C07332=1146.015,329.799,-77.371,-176.675,8.921,148.819
C07333=1146.011,330.047,-77.404,-176.672,8.925,148.820
C07334=1146.007,330.294,-77.436,-176.670,8.928,148.820
C07335=1146.003,330.542,-77.470,-176.667,8.932,148.820
C07336=1145.999,330.789,-77.503,-176.665,8.936,148.820
C07337=1145.995,331.037,-77.536,-176.662,8.940,148.821
C07338=1145.991,331.285,-77.569,-176.659,8.943,148.821
C07339=1145.986,331.533,-77.602,-176.657,8.947,148.821
C07340=1145.982,331.780,-77.635,-176.654,8.950,148.821
C07341=1145.978,332.028,-77.669,-176.651,8.954,148.821
C07342=1145.974,332.276,-77.702,-176.649,8.958,148.822
C07343=1145.970,332.524,-77.735,-176.646,8.962,148.822
C07344=1145.966,332.771,-77.768,-176.644,8.965,148.822
C07345=1145.962,333.020,-77.802,-176.641,8.969,148.823
C07346=1145.958,333.267,-77.835,-176.639,8.973,148.823
C07347=1145.954,333.515,-77.868,-176.637,8.976,148.823
C07348=1145.950,333.763,-77.901,-176.634,8.980,148.823
C07349=1145.946,334.010,-77.935,-176.631,8.983,148.823
C07350=1145.942,334.258,-77.968,-176.628,8.987,148.824
C07351=1145.938,334.505,-78.001,-176.627,8.991,148.824
C07352=1145.934,334.753,-78.034,-176.624,8.995,148.824
C07353=1145.930,335.002,-78.068,-176.621,8.998,148.824
C07354=1145.926,335.249,-78.102,-176.618,9.002,148.825
C07355=1145.922,335.496,-78.135,-176.615,9.006,148.825
C07356=1145.918,335.744,-78.168,-176.613,9.010,148.825
C07357=1145.913,335.992,-78.202,-176.611,9.014,148.826
C07358=1145.909,336.239,-78.236,-176.608,9.017,148.826
C07359=1145.906,336.488,-78.269,-176.605,9.021,148.826
C07360=1145.902,336.735,-78.302,-176.603,9.025,148.826
C07361=1145.897,336.983,-78.336,-176.600,9.029,148.826
C07362=1145.894,337.230,-78.369,-176.598,9.032,148.827
C07363=1145.889,337.478,-78.403,-176.595,9.036,148.827
C07364=1145.885,337.727,-78.437,-176.593,9.040,148.827
C07365=1145.881,337.974,-78.471,-176.590,9.044,148.828
C07366=1145.877,338.222,-78.504,-176.588,9.047,148.828
C07367=1145.873,338.469,-78.538,-176.585,9.051,148.828
C07368=1145.869,338.716,-78.571,-176.583,9.055,148.828
C07369=1145.864,338.997,-78.609,-176.580,9.059,148.829
C07370=1145.860,339.277,-78.647,-176.577,9.064,148.829
C07371=1145.856,339.558,-78.686,-176.574,9.068,148.829
C07372=1145.851,339.839,-78.724,-176.571,9.072,148.830
C07373=1145.847,340.086,-78.757,-176.569,9.075,148.830
C07374=1145.843,340.333,-78.791,-176.566,9.080,148.830
C07375=1145.838,340.581,-78.825,-176.564,9.083,148.830
C07376=1145.835,340.829,-78.859,-176.561,9.087,148.831
C07377=1145.831,341.076,-78.893,-176.558,9.091,148.831
C07378=1145.827,341.324,-78.926,-176.556,9.095,148.831
C07379=1145.823,341.572,-78.961,-176.553,9.099,148.832
C07380=1145.819,341.820,-78.994,-176.551,9.102,148.832
C07381=1145.815,342.067,-79.028,-176.548,9.106,148.832
C07382=1145.810,342.314,-79.062,-176.546,9.110,148.832
C07383=1145.807,342.563,-79.096,-176.543,9.114,148.833
C07384=1145.802,342.810,-79.130,-176.541,9.117,148.833
C07385=1145.799,343.057,-79.164,-176.538,9.121,148.833
C07386=1145.795,343.306,-79.198,-176.536,9.126,148.834
C07387=1145.790,343.553,-79.232,-176.533,9.129,148.834
C07388=1145.787,343.800,-79.266,-176.530,9.133,148.834
C07389=1145.783,344.049,-79.300,-176.528,9.137,148.834
C07390=1145.778,344.296,-79.334,-176.525,9.141,148.835
C07391=1145.775,344.543,-79.368,-176.523,9.144,148.835
C07392=1145.771,344.791,-79.403,-176.521,9.148,148.835
C07393=1145.767,345.039,-79.436,-176.518,9.152,148.836
C07394=1145.762,345.287,-79.470,-176.515,9.156,148.836
C07395=1145.759,345.534,-79.505,-176.513,9.160,148.836
C07396=1145.754,345.782,-79.539,-176.511,9.163,148.836
C07397=1145.751,346.030,-79.573,-176.508,9.167,148.837
C07398=1145.746,346.277,-79.608,-176.506,9.171,148.837
C07399=1145.742,346.525,-79.641,-176.503,9.175,148.837
C07400=1145.738,346.773,-79.676,-176.500,9.179,148.838
C07401=1145.734,347.020,-79.710,-176.498,9.183,148.838
C07402=1145.730,347.268,-79.745,-176.495,9.187,148.838
C07403=1145.727,347.515,-79.778,-176.493,9.190,148.838
C07404=1145.722,347.763,-79.813,-176.490,9.195,148.839
C07405=1145.719,348.011,-79.847,-176.487,9.199,148.839
C07406=1145.714,348.258,-79.882,-176.485,9.202,148.839
C07407=1145.711,348.506,-79.916,-176.483,9.206,148.840
C07408=1145.706,348.753,-79.950,-176.480,9.210,148.840
C07409=1145.702,349.001,-79.985,-176.477,9.214,148.840
C07410=1145.699,349.248,-80.019,-176.475,9.217,148.841
C07411=1145.695,349.497,-80.054,-176.473,9.221,148.841
C07412=1145.691,349.744,-80.088,-176.470,9.226,148.841
C07413=1145.687,349.992,-80.123,-176.468,9.229,148.842
C07414=1145.682,350.239,-80.157,-176.465,9.233,148.842
C07415=1145.679,350.486,-80.192,-176.462,9.237,148.842
C07416=1145.675,350.734,-80.226,-176.460,9.241,148.843
C07417=1145.671,350.982,-80.261,-176.457,9.245,148.843
C07418=1145.667,351.229,-80.295,-176.455,9.248,148.843
C07419=1145.663,351.477,-80.330,-176.452,9.252,148.843
C07420=1145.658,351.725,-80.364,-176.450,9.257,148.844
C07421=1145.656,351.972,-80.399,-176.447,9.260,148.844
C07422=1145.651,352.219,-80.434,-176.445,9.264,148.845
C07423=1145.647,352.467,-80.469,-176.443,9.268,148.845
C07424=1145.643,352.714,-80.503,-176.440,9.272,148.845
C07425=1145.640,352.962,-80.538,-176.437,9.276,148.846
C07426=1145.635,353.209,-80.573,-176.435,9.279,148.846
C07427=1145.631,353.457,-80.607,-176.432,9.284,148.846
C07428=1145.627,353.704,-80.642,-176.429,9.288,148.846
C07429=1145.623,353.952,-80.677,-176.428,9.292,148.847
C07430=1145.620,354.200,-80.712,-176.425,9.296,148.847
C07431=1145.615,354.447,-80.747,-176.422,9.300,148.848
C07432=1145.612,354.695,-80.781,-176.420,9.303,148.848
C07433=1145.607,354.942,-80.816,-176.417,9.308,148.848
C07434=1145.604,355.190,-80.851,-176.415,9.311,148.848
C07435=1145.600,355.438,-80.886,-176.412,9.315,148.849
C07436=1145.596,355.685,-80.921,-176.410,9.319,148.849
C07437=1145.592,355.932,-80.955,-176.407,9.323,148.849
C07438=1145.588,356.180,-80.990,-176.405,9.327,148.850
C07439=1145.584,356.427,-81.025,-176.402,9.331,148.850
C07440=1145.580,356.675,-81.060,-176.400,9.335,148.850
C07441=1145.576,356.922,-81.095,-176.397,9.339,148.851
C07442=1145.572,357.170,-81.130,-176.394,9.343,148.851
C07443=1145.568,357.418,-81.166,-176.392,9.346,148.851
C07444=1145.564,357.665,-81.201,-176.390,9.351,148.852
C07445=1145.561,357.912,-81.235,-176.387,9.355,148.852
C07446=1145.557,358.160,-81.271,-176.385,9.359,148.853
C07447=1145.553,358.407,-81.305,-176.382,9.363,148.853
C07448=1145.549,358.655,-81.341,-176.379,9.367,148.853
C07449=1145.545,358.902,-81.376,-176.377,9.370,148.853
C07450=1145.541,359.150,-81.411,-176.375,9.375,148.854
C07451=1145.537,359.397,-81.446,-176.372,9.379,148.854
C07452=1145.533,359.645,-81.482,-176.369,9.383,148.855
C07453=1145.529,359.893,-81.517,-176.367,9.386,148.855
C07454=1145.525,360.140,-81.552,-176.364,9.391,148.855
C07455=1145.521,360.387,-81.587,-176.361,9.395,148.856
C07456=1145.517,360.635,-81.622,-176.359,9.399,148.856
C07457=1145.513,360.882,-81.657,-176.357,9.403,148.856
C07458=1145.509,361.130,-81.693,-176.354,9.407,148.857
C07459=1145.506,361.377,-81.729,-176.351,9.411,148.857
C07460=1145.502,361.625,-81.764,-176.349,9.415,148.857
C07461=1145.498,361.872,-81.799,-176.346,9.419,148.858
C07462=1145.494,362.120,-81.834,-176.343,9.423,148.858
C07463=1145.490,362.367,-81.870,-176.341,9.427,148.858
C07464=1145.487,362.615,-81.905,-176.338,9.431,148.859
C07465=1145.483,362.862,-81.941,-176.336,9.435,148.859
C07466=1145.479,363.109,-81.976,-176.333,9.439,148.859
C07467=1145.475,363.356,-82.011,-176.331,9.443,148.860
C07468=1145.471,363.604,-82.048,-176.328,9.447,148.860
C07469=1145.467,363.852,-82.082,-176.325,9.452,148.861
C07470=1145.463,364.100,-82.118,-176.322,9.456,148.861
C07471=1145.459,364.347,-82.153,-176.320,9.459,148.861
C07472=1145.455,364.594,-82.189,-176.317,9.463,148.861
C07473=1145.451,364.877,-82.230,-176.314,9.469,148.862
C07474=1145.446,365.161,-82.270,-176.311,9.473,148.862
C07475=1145.442,365.444,-82.311,-176.308,9.478,148.863
C07476=1145.437,365.728,-82.352,-176.306,9.482,148.863
C07477=1145.433,365.975,-82.388,-176.303,9.486,148.864
C07478=1145.429,366.223,-82.424,-176.300,9.491,148.864
C07479=1145.426,366.470,-82.459,-176.298,9.495,148.864
C07480=1145.422,366.717,-82.495,-176.295,9.499,148.865
C07481=1145.419,366.965,-82.531,-176.292,9.503,148.865
C07482=1145.414,367.213,-82.567,-176.290,9.508,148.865
C07483=1145.410,367.459,-82.602,-176.287,9.512,148.866
C07484=1145.406,367.707,-82.638,-176.284,9.516,148.866
C07485=1145.402,367.955,-82.674,-176.282,9.519,148.866
C07486=1145.399,368.202,-82.710,-176.279,9.524,148.867
C07487=1145.395,368.449,-82.746,-176.277,9.528,148.867
C07488=1145.390,368.697,-82.782,-176.274,9.532,148.868
C07489=1145.387,368.944,-82.817,-176.271,9.537,148.868
C07490=1145.383,369.191,-82.854,-176.269,9.541,148.869
C07491=1145.379,369.439,-82.890,-176.266,9.545,148.869
C07492=1145.375,369.687,-82.925,-176.264,9.550,148.869
C07493=1145.372,369.934,-82.961,-176.261,9.554,148.870
C07494=1145.368,370.181,-82.998,-176.259,9.557,148.870
C07495=1145.363,370.428,-83.033,-176.256,9.562,148.870
C07496=1145.360,370.675,-83.069,-176.254,9.566,148.871
C07497=1145.356,370.923,-83.105,-176.251,9.570,148.871
C07498=1145.352,371.170,-83.141,-176.248,9.575,148.872
C07499=1145.348,371.417,-83.178,-176.246,9.579,148.872
C07500=1145.344,371.665,-83.213,-176.243,9.583,148.873
C07501=1145.341,371.912,-83.250,-176.241,9.587,148.873
C07502=1145.336,372.160,-83.286,-176.238,9.591,148.873
C07503=1145.333,372.407,-83.322,-176.236,9.595,148.874
C07504=1145.329,372.654,-83.358,-176.233,9.600,148.874
C07505=1145.325,372.901,-83.394,-176.231,9.604,148.875
C07506=1145.321,373.149,-83.431,-176.228,9.608,148.875
C07507=1145.318,373.396,-83.467,-176.227,9.612,148.876
C07508=1145.313,373.644,-83.503,-176.224,9.616,148.876
C07509=1145.310,373.891,-83.539,-176.222,9.621,148.876
C07510=1145.305,374.138,-83.575,-176.219,9.625,148.877
C07511=1145.303,374.386,-83.612,-176.217,9.629,148.877
C07512=1145.298,374.634,-83.648,-176.215,9.633,148.878
C07513=1145.295,374.881,-83.684,-176.212,9.638,148.878
C07514=1145.291,375.128,-83.721,-176.210,9.641,148.879
C07515=1145.287,375.375,-83.757,-176.208,9.646,148.879
C07516=1145.283,375.623,-83.794,-176.205,9.650,148.880
C07517=1145.279,375.870,-83.831,-176.204,9.654,148.880
C07518=1145.275,376.117,-83.866,-176.201,9.658,148.881
C07519=1145.271,376.364,-83.903,-176.199,9.662,148.881
C07520=1145.268,376.611,-83.939,-176.197,9.666,148.882
C07521=1145.264,376.859,-83.976,-176.195,9.670,148.882
C07522=1145.259,377.106,-84.012,-176.193,9.674,148.883
C07523=1145.256,377.353,-84.048,-176.191,9.678,148.883
C07524=1145.253,377.601,-84.086,-176.189,9.683,148.884
C07525=1145.248,377.848,-84.123,-176.187,9.686,148.884
C07526=1145.245,378.095,-84.159,-176.185,9.691,148.885
C07527=1145.241,378.343,-84.195,-176.183,9.695,148.886
C07528=1145.237,378.590,-84.232,-176.181,9.698,148.886
C07529=1145.233,378.837,-84.268,-176.180,9.702,148.887
C07530=1145.229,379.084,-84.305,-176.178,9.707,148.887
C07531=1145.225,379.331,-84.342,-176.176,9.711,148.888
C07532=1145.222,379.579,-84.378,-176.174,9.714,148.888
C07533=1145.218,379.826,-84.415,-176.173,9.718,148.889
C07534=1145.214,380.074,-84.451,-176.171,9.722,148.889
C07535=1145.210,380.321,-84.488,-176.170,9.726,148.890
C07536=1145.206,380.568,-84.525,-176.168,9.730,148.891
C07537=1145.202,380.815,-84.561,-176.167,9.734,148.891
C07538=1145.199,381.063,-84.599,-176.165,9.738,148.892
C07539=1145.195,381.310,-84.635,-176.164,9.742,148.893
C07540=1145.191,381.557,-84.672,-176.162,9.746,148.893
C07541=1145.187,381.804,-84.709,-176.162,9.749,148.894
C07542=1145.183,382.052,-84.745,-176.160,9.752,148.894
C07543=1145.179,382.299,-84.782,-176.159,9.757,148.895
C07544=1145.176,382.546,-84.819,-176.158,9.760,148.896
C07545=1145.172,382.794,-84.856,-176.157,9.764,148.896
C07546=1145.168,383.041,-84.893,-176.156,9.767,148.897
C07547=1145.164,383.288,-84.930,-176.155,9.770,148.898
C07548=1145.160,383.535,-84.966,-176.154,9.774,148.898
C07549=1145.157,383.783,-85.003,-176.153,9.777,148.899
C07550=1145.153,384.029,-85.041,-176.153,9.781,148.900
C07551=1145.149,384.277,-85.077,-176.152,9.784,148.900
C07552=1145.145,384.524,-85.114,-176.152,9.787,148.901
C07553=1145.142,384.772,-85.152,-176.151,9.791,148.902
C07554=1145.138,385.019,-85.188,-176.150,9.794,148.903
C07555=1145.134,385.266,-85.225,-176.150,9.797,148.903
C07556=1145.130,385.513,-85.261,-176.149,9.801,148.904
C07557=1145.126,385.760,-85.298,-176.149,9.804,148.905
C07558=1145.123,386.008,-85.336,-176.149,9.807,148.906
C07559=1145.119,386.255,-85.373,-176.148,9.810,148.906
C07560=1145.115,386.502,-85.410,-176.149,9.813,148.907
C07561=1145.111,386.749,-85.446,-176.148,9.816,148.908
C07562=1145.108,386.996,-85.483,-176.149,9.819,148.909
C07563=1145.104,387.244,-85.520,-176.149,9.821,148.909
C07564=1145.100,387.491,-85.557,-176.149,9.825,148.910
C07565=1145.096,387.737,-85.595,-176.149,9.828,148.911
C07566=1145.092,387.985,-85.632,-176.149,9.830,148.912
C07567=1145.088,388.233,-85.669,-176.149,9.833,148.913
C07568=1145.084,388.480,-85.706,-176.149,9.836,148.913
C07569=1145.081,388.727,-85.742,-176.150,9.838,148.914
C07570=1145.078,388.974,-85.780,-176.150,9.841,148.915
C07571=1145.073,389.221,-85.817,-176.151,9.844,148.916
C07572=1145.069,389.468,-85.854,-176.151,9.846,148.916
C07573=1145.066,389.716,-85.891,-176.151,9.849,148.917
C07574=1145.062,389.963,-85.928,-176.152,9.852,148.918
C07575=1145.058,390.210,-85.965,-176.152,9.855,148.919
C07576=1145.054,390.457,-86.002,-176.152,9.858,148.920
C07577=1145.050,390.745,-86.045,-176.153,9.860,148.921
C07578=1145.046,391.031,-86.088,-176.154,9.863,148.922
C07579=1145.041,391.318,-86.131,-176.155,9.866,148.923
C07580=1145.037,391.605,-86.174,-176.155,9.869,148.924
C07581=1145.033,391.852,-86.211,-176.156,9.872,148.924
C07582=1145.029,392.099,-86.248,-176.157,9.874,148.925
C07583=1145.026,392.347,-86.285,-176.157,9.876,148.926
C07584=1145.022,392.594,-86.322,-176.159,9.879,148.927
C07585=1145.018,392.841,-86.360,-176.160,9.881,148.928
C07586=1145.014,393.088,-86.397,-176.160,9.883,148.929
C07587=1145.010,393.336,-86.434,-176.161,9.885,148.929
C07588=1145.006,393.583,-86.471,-176.162,9.887,148.930
C07589=1145.002,393.830,-86.508,-176.162,9.890,148.931
C07590=1145.000,394.077,-86.545,-176.164,9.892,148.932
C07591=1144.995,394.324,-86.582,-176.165,9.894,148.933
C07592=1144.991,394.571,-86.619,-176.166,9.896,148.934
C07593=1144.988,394.818,-86.656,-176.166,9.899,148.934
C07594=1144.984,395.066,-86.693,-176.167,9.901,148.935
C07595=1144.980,395.313,-86.730,-176.168,9.903,148.936
C07596=1144.976,395.560,-86.767,-176.170,9.905,148.937
C07597=1144.972,395.807,-86.805,-176.171,9.907,148.938
C07598=1144.969,396.055,-86.842,-176.172,9.910,148.939
C07599=1144.965,396.302,-86.879,-176.173,9.912,148.939
C07600=1144.960,396.549,-86.916,-176.174,9.914,148.940
C07601=1144.957,396.796,-86.954,-176.175,9.916,148.941
C07602=1144.953,397.044,-86.990,-176.176,9.918,148.942
C07603=1144.949,397.291,-87.027,-176.177,9.920,148.943
C07604=1144.945,397.538,-87.064,-176.178,9.922,148.944
C07605=1144.943,397.785,-87.101,-176.179,9.924,148.944
C07606=1144.938,398.032,-87.138,-176.181,9.926,148.945
C07607=1144.934,398.279,-87.175,-176.182,9.928,148.946
C07608=1144.931,398.527,-87.212,-176.183,9.930,148.947
C07609=1144.927,398.774,-87.250,-176.184,9.932,148.948
C07610=1144.923,399.021,-87.287,-176.185,9.934,148.949
C07611=1144.919,399.268,-87.324,-176.186,9.936,148.950
C07612=1144.916,399.515,-87.362,-176.187,9.938,148.950
C07613=1144.912,399.763,-87.398,-176.188,9.940,148.951
C07614=1144.907,400.010,-87.435,-176.190,9.942,148.952
C07615=1144.903,400.257,-87.472,-176.191,9.944,148.953
C07616=1144.900,400.504,-87.510,-176.192,9.946,148.954
C07617=1144.896,400.751,-87.547,-176.193,9.948,148.954
C07618=1144.892,400.999,-87.584,-176.194,9.950,148.955
C07619=1144.889,401.247,-87.621,-176.195,9.952,148.956
C07620=1144.885,401.493,-87.658,-176.196,9.954,148.957
C07621=1144.881,401.740,-87.695,-176.198,9.956,148.958
C07622=1144.877,401.987,-87.732,-176.199,9.957,148.959
C07623=1144.874,402.235,-87.769,-176.200,9.959,148.959
C07624=1144.870,402.482,-87.807,-176.201,9.961,148.960
C07625=1144.866,402.729,-87.843,-176.203,9.964,148.961
C07626=1144.862,402.976,-87.880,-176.203,9.965,148.962
C07627=1144.858,403.224,-87.918,-176.204,9.967,148.963
C07628=1144.855,403.471,-87.955,-176.206,9.969,148.963
C07629=1144.850,403.718,-87.992,-176.207,9.971,148.964
C07630=1144.847,403.966,-88.029,-176.208,9.973,148.965
C07631=1144.843,404.213,-88.066,-176.209,9.975,148.966
C07632=1144.839,404.459,-88.104,-176.210,9.977,148.967
C07633=1144.835,404.707,-88.140,-176.211,9.979,148.967
C07634=1144.831,404.954,-88.178,-176.213,9.981,148.968
C07635=1144.828,405.201,-88.215,-176.213,9.983,148.969
C07636=1144.824,405.448,-88.252,-176.215,9.984,148.970
C07637=1144.821,405.696,-88.289,-176.216,9.986,148.971
C07638=1144.817,405.943,-88.326,-176.217,9.988,148.971
C07639=1144.813,406.190,-88.363,-176.218,9.990,148.972
C07640=1144.809,406.437,-88.400,-176.219,9.992,148.973
C07641=1144.805,406.685,-88.437,-176.220,9.994,148.974
C07642=1144.801,406.932,-88.474,-176.221,9.996,148.975
C07643=1144.797,407.178,-88.512,-176.222,9.998,148.975
C07644=1144.793,407.426,-88.549,-176.223,10.000,148.976
C07645=1144.790,407.673,-88.586,-176.224,10.002,148.977
C07646=1144.786,407.921,-88.623,-176.226,10.003,148.978
C07647=1144.782,408.167,-88.660,-176.227,10.005,148.978
C07648=1144.779,408.415,-88.697,-176.228,10.007,148.979
C07649=1144.775,408.662,-88.734,-176.228,10.009,148.980
C07650=1144.771,408.909,-88.771,-176.229,10.011,148.981
C07651=1144.767,409.156,-88.808,-176.231,10.013,148.982
C07652=1144.764,409.404,-88.845,-176.231,10.015,148.982
C07653=1144.760,409.651,-88.882,-176.232,10.017,148.983
C07654=1144.756,409.897,-88.920,-176.233,10.019,148.984
C07655=1144.752,410.145,-88.957,-176.234,10.021,148.985
C07656=1144.748,410.392,-88.994,-176.235,10.023,148.985
C07657=1144.744,410.640,-89.031,-176.236,10.025,148.986
C07658=1144.740,410.886,-89.068,-176.237,10.027,148.987
C07659=1144.737,411.134,-89.106,-176.238,10.029,148.988
C07660=1144.733,411.381,-89.142,-176.238,10.031,148.988
C07661=1144.729,411.629,-89.179,-176.239,10.033,148.989
C07662=1144.725,411.875,-89.217,-176.240,10.035,148.990
C07663=1144.721,412.123,-89.254,-176.241,10.037,148.991
C07664=1144.717,412.370,-89.291,-176.242,10.039,148.991
C07665=1144.713,412.617,-89.328,-176.243,10.041,148.992
C07666=1144.710,412.865,-89.366,-176.244,10.043,148.993
C07667=1144.707,413.112,-89.402,-176.244,10.045,148.994
C07668=1144.703,413.359,-89.439,-176.245,10.047,148.994
C07669=1144.699,413.605,-89.476,-176.246,10.049,148.995
C07670=1144.695,413.853,-89.514,-176.247,10.052,148.996
C07671=1144.691,414.100,-89.550,-176.247,10.053,148.997
C07672=1144.687,414.348,-89.587,-176.248,10.055,148.997
C07673=1144.684,414.595,-89.625,-176.249,10.057,148.998
C07674=1144.680,414.842,-89.662,-176.250,10.059,148.999
C07675=1144.677,415.089,-89.699,-176.250,10.062,149.000
C07676=1144.676,415.337,-89.736,-176.251,10.064,149.000
C07677=1144.675,415.580,-89.772,-176.252,10.066,149.001
C07678=1144.675,415.824,-89.809,-176.253,10.067,149.002
C07679=1144.675,416.068,-89.845,-176.253,10.069,149.002
C07680=1144.676,416.312,-89.881,-176.253,10.072,149.003
C07681=1144.677,416.555,-89.916,-176.254,10.073,149.004
C07682=1144.679,416.799,-89.953,-176.255,10.075,149.004
C07683=1144.682,417.042,-89.989,-176.256,10.077,149.005
C07684=1144.686,417.285,-90.024,-176.256,10.079,149.006
C07685=1144.266,417.287,-90.074,-176.258,10.090,149.009
C07686=1144.263,417.042,-90.038,-176.257,10.088,149.008
C07687=1144.259,416.797,-90.002,-176.257,10.086,149.008
C07688=1144.256,416.552,-89.966,-176.257,10.084,149.007
C07689=1144.255,416.307,-89.929,-176.256,10.082,149.006
C07690=1144.254,416.062,-89.893,-176.255,10.081,149.006
C07691=1144.254,415.816,-89.857,-176.254,10.079,149.005
C07692=1144.254,415.571,-89.821,-176.253,10.077,149.004
C07693=1144.255,415.325,-89.784,-176.253,10.074,149.004
C07694=1144.258,415.078,-89.747,-176.252,10.072,149.003
C07695=1144.260,414.831,-89.710,-176.252,10.070,149.002
C07696=1144.263,414.583,-89.673,-176.251,10.068,149.001
C07697=1144.267,414.336,-89.636,-176.250,10.067,149.001
C07698=1144.270,414.089,-89.598,-176.249,10.064,149.000
C07699=1144.274,413.842,-89.561,-176.249,10.062,148.999
C07700=1144.278,413.594,-89.525,-176.248,10.060,148.998
C07701=1144.282,413.347,-89.487,-176.247,10.058,148.998
C07702=1144.286,413.100,-89.450,-176.246,10.056,148.997
C07703=1144.290,412.853,-89.413,-176.245,10.054,148.996
C07704=1144.294,412.606,-89.375,-176.245,10.051,148.995
C07705=1144.297,412.358,-89.338,-176.244,10.050,148.995
C07706=1144.301,412.111,-89.301,-176.243,10.048,148.994
C07707=1144.305,411.864,-89.264,-176.242,10.046,148.993
C07708=1144.308,411.617,-89.226,-176.241,10.044,148.992
C07709=1144.313,411.369,-89.190,-176.240,10.042,148.992
C07710=1144.317,411.122,-89.153,-176.240,10.040,148.991
C07711=1144.320,410.876,-89.115,-176.238,10.038,148.990
C07712=1144.323,410.628,-89.079,-176.237,10.036,148.989
C07713=1144.327,410.381,-89.042,-176.237,10.034,148.989
C07714=1144.331,410.134,-89.005,-176.236,10.032,148.988
C07715=1144.335,409.886,-88.967,-176.235,10.030,148.987
C07716=1144.339,409.639,-88.930,-176.234,10.028,148.986
C07717=1144.343,409.392,-88.893,-176.233,10.026,148.986
C07718=1144.347,409.145,-88.856,-176.232,10.024,148.985
C07719=1144.350,408.898,-88.818,-176.231,10.022,148.984
C07720=1144.354,408.650,-88.782,-176.230,10.020,148.983
C07721=1144.358,408.403,-88.745,-176.229,10.018,148.982
C07722=1144.361,408.156,-88.707,-176.228,10.016,148.982
C07723=1144.366,407.909,-88.670,-176.227,10.014,148.981
C07724=1144.370,407.662,-88.633,-176.226,10.012,148.980
C07725=1144.374,407.414,-88.596,-176.225,10.010,148.979
C07726=1144.377,407.167,-88.558,-176.224,10.008,148.978
C07727=1144.381,406.920,-88.521,-176.223,10.006,148.978
C07728=1144.385,406.673,-88.485,-176.222,10.004,148.977
C07729=1144.389,406.426,-88.447,-176.221,10.002,148.976
C07730=1144.392,406.179,-88.410,-176.220,10.000,148.975
C07731=1144.396,405.931,-88.373,-176.218,9.999,148.975
C07732=1144.400,405.684,-88.337,-176.217,9.997,148.974
C07733=1144.403,405.437,-88.299,-176.216,9.995,148.973
C07734=1144.407,405.190,-88.262,-176.215,9.993,148.972
C07735=1144.411,404.942,-88.225,-176.214,9.991,148.971
C07736=1144.415,404.695,-88.188,-176.213,9.989,148.971
C07737=1144.418,404.448,-88.150,-176.212,9.987,148.970
C07738=1144.423,404.201,-88.113,-176.211,9.985,148.969
C07739=1144.427,403.954,-88.076,-176.209,9.984,148.968
C07740=1144.430,403.706,-88.038,-176.208,9.982,148.967
C07741=1144.434,403.459,-88.002,-176.207,9.979,148.966
C07742=1144.438,403.212,-87.965,-176.206,9.977,148.966
C07743=1144.442,402.965,-87.928,-176.205,9.976,148.965
C07744=1144.445,402.718,-87.890,-176.204,9.974,148.964
C07745=1144.449,402.470,-87.853,-176.203,9.972,148.963
C07746=1144.453,402.223,-87.817,-176.202,9.970,148.963
C07747=1144.456,401.976,-87.780,-176.200,9.968,148.962
C07748=1144.460,401.729,-87.742,-176.199,9.966,148.961
C07749=1144.464,401.482,-87.705,-176.198,9.964,148.960
C07750=1144.468,401.235,-87.668,-176.197,9.962,148.959
C07751=1144.471,400.987,-87.630,-176.196,9.960,148.958
C07752=1144.476,400.740,-87.594,-176.194,9.959,148.958
C07753=1144.480,400.493,-87.557,-176.193,9.957,148.957
C07754=1144.483,400.245,-87.519,-176.192,9.955,148.956
C07755=1144.487,399.999,-87.482,-176.191,9.953,148.955
C07756=1144.491,399.751,-87.445,-176.190,9.950,148.954
C07757=1144.495,399.504,-87.408,-176.189,9.948,148.953
C07758=1144.499,399.256,-87.371,-176.188,9.946,148.953
C07759=1144.502,399.010,-87.333,-176.187,9.944,148.952
C07760=1144.506,398.762,-87.297,-176.186,9.942,148.951
C07761=1144.510,398.515,-87.259,-176.184,9.941,148.950
C07762=1144.514,398.268,-87.222,-176.183,9.939,148.949
C07763=1144.518,398.021,-87.185,-176.182,9.937,148.948
C07764=1144.521,397.774,-87.149,-176.181,9.935,148.948
C07765=1144.525,397.526,-87.111,-176.180,9.933,148.947
C07766=1144.528,397.279,-87.074,-176.178,9.931,148.946
C07767=1144.533,397.032,-87.037,-176.177,9.929,148.945
C07768=1144.537,396.785,-87.000,-176.176,9.927,148.944
C07769=1144.540,396.537,-86.963,-176.175,9.924,148.943
C07770=1144.544,396.291,-86.925,-176.174,9.922,148.943
C07771=1144.548,396.043,-86.888,-176.173,9.920,148.942
C07772=1144.552,395.796,-86.851,-176.172,9.918,148.941
C07773=1144.555,395.549,-86.814,-176.171,9.916,148.940
C07774=1144.559,395.302,-86.777,-176.170,9.913,148.939
C07775=1144.563,395.055,-86.740,-176.169,9.911,148.938
C07776=1144.567,394.807,-86.703,-176.168,9.909,148.938
C07777=1144.571,394.560,-86.665,-176.167,9.907,148.937
C07778=1144.575,394.313,-86.628,-176.166,9.905,148.936
C07779=1144.578,394.065,-86.591,-176.165,9.903,148.935
C07780=1144.582,393.818,-86.554,-176.164,9.900,148.934
C07781=1144.586,393.572,-86.517,-176.163,9.898,148.933
C07782=1144.590,393.324,-86.480,-176.162,9.896,148.933
C07783=1144.593,393.077,-86.443,-176.162,9.893,148.932
C07784=1144.597,392.830,-86.406,-176.160,9.891,148.931
C07785=1144.601,392.583,-86.369,-176.159,9.889,148.930
C07786=1144.604,392.335,-86.331,-176.159,9.887,148.929
C07787=1144.609,392.088,-86.295,-176.158,9.884,148.928
C07788=1144.612,391.841,-86.257,-176.158,9.882,148.928
C07789=1144.616,391.594,-86.220,-176.157,9.880,148.927
C07790=1144.620,391.306,-86.177,-176.156,9.877,148.926
C07791=1144.625,391.020,-86.134,-176.155,9.873,148.925
C07792=1144.629,390.733,-86.091,-176.155,9.871,148.924
C07793=1144.634,390.445,-86.048,-176.154,9.868,148.923
C07794=1144.637,390.199,-86.011,-176.153,9.866,148.922
C07795=1144.641,389.951,-85.974,-176.153,9.863,148.921
C07796=1144.645,389.704,-85.937,-176.152,9.860,148.921
C07797=1144.649,389.457,-85.900,-176.152,9.857,148.920
C07798=1144.653,389.210,-85.863,-176.152,9.855,148.919
C07799=1144.656,388.962,-85.825,-176.151,9.852,148.918
C07800=1144.660,388.715,-85.789,-176.151,9.849,148.917
C07801=1144.664,388.468,-85.752,-176.151,9.846,148.916
C07802=1144.668,388.221,-85.715,-176.151,9.844,148.916
C07803=1144.672,387.974,-85.677,-176.150,9.841,148.915
C07804=1144.675,387.727,-85.641,-176.150,9.838,148.914
C07805=1144.679,387.480,-85.604,-176.150,9.836,148.913
C07806=1144.683,387.232,-85.567,-176.150,9.832,148.913
C07807=1144.687,386.984,-85.530,-176.150,9.830,148.912
C07808=1144.690,386.738,-85.492,-176.150,9.827,148.911
C07809=1144.694,386.491,-85.455,-176.150,9.824,148.910
C07810=1144.699,386.243,-85.418,-176.150,9.821,148.910
C07811=1144.701,385.996,-85.382,-176.151,9.818,148.909
C07812=1144.705,385.749,-85.345,-176.151,9.814,148.908
C07813=1144.709,385.502,-85.308,-176.151,9.812,148.907
C07814=1144.714,385.254,-85.271,-176.151,9.808,148.907
C07815=1144.717,385.007,-85.233,-176.152,9.805,148.906
C07816=1144.721,384.760,-85.196,-176.152,9.802,148.905
C07817=1144.725,384.513,-85.160,-176.153,9.798,148.904
C07818=1144.728,384.266,-85.123,-176.153,9.795,148.904
C07819=1144.732,384.018,-85.086,-176.154,9.792,148.903
C07820=1144.736,383.771,-85.049,-176.155,9.789,148.902
C07821=1144.740,383.524,-85.012,-176.155,9.785,148.902
C07822=1144.744,383.276,-84.975,-176.157,9.781,148.901
C07823=1144.748,383.029,-84.939,-176.157,9.778,148.900
C07824=1144.751,382.782,-84.902,-176.158,9.775,148.900
C07825=1144.755,382.535,-84.864,-176.160,9.771,148.899
C07826=1144.759,382.288,-84.828,-176.160,9.768,148.898
C07827=1144.763,382.041,-84.791,-176.162,9.764,148.898
C07828=1144.766,381.793,-84.754,-176.163,9.760,148.897
C07829=1144.770,381.546,-84.717,-176.164,9.757,148.897
C07830=1144.774,381.299,-84.680,-176.166,9.753,148.896
C07831=1144.778,381.051,-84.643,-176.167,9.749,148.895
C07832=1144.782,380.804,-84.607,-176.168,9.745,148.894
C07833=1144.785,380.557,-84.570,-176.170,9.741,148.894
C07834=1144.789,380.309,-84.534,-176.172,9.737,148.893
C07835=1144.793,380.062,-84.497,-176.173,9.733,148.893
C07836=1144.797,379.815,-84.461,-176.175,9.730,148.892
C07837=1144.801,379.568,-84.424,-176.176,9.726,148.892
C07838=1144.805,379.320,-84.387,-176.178,9.722,148.891
C07839=1144.809,379.073,-84.350,-176.180,9.718,148.891
C07840=1144.812,378.826,-84.314,-176.182,9.714,148.890
C07841=1144.816,378.578,-84.277,-176.183,9.710,148.889
C07842=1144.820,378.331,-84.240,-176.185,9.706,148.889
C07843=1144.824,378.084,-84.204,-176.187,9.701,148.888
C07844=1144.828,377.837,-84.167,-176.189,9.698,148.888
C07845=1144.832,377.589,-84.131,-176.191,9.694,148.887
C07846=1144.835,377.343,-84.094,-176.193,9.690,148.887
C07847=1144.839,377.095,-84.057,-176.194,9.686,148.886
C07848=1144.844,376.848,-84.021,-176.197,9.681,148.886
C07849=1144.846,376.600,-83.985,-176.199,9.678,148.885
C07850=1144.850,376.353,-83.948,-176.201,9.673,148.885
C07851=1144.855,376.106,-83.911,-176.203,9.669,148.884
C07852=1144.858,375.858,-83.875,-176.205,9.665,148.884
C07853=1144.862,375.611,-83.839,-176.208,9.661,148.883
C07854=1144.866,375.364,-83.802,-176.210,9.657,148.883
C07855=1144.870,375.116,-83.766,-176.212,9.652,148.882
C07856=1144.873,374.869,-83.730,-176.214,9.648,148.882
C07857=1144.878,374.622,-83.693,-176.216,9.644,148.881
C07858=1144.881,374.375,-83.657,-176.219,9.640,148.881
C07859=1144.885,374.127,-83.621,-176.221,9.636,148.880
C07860=1144.889,373.880,-83.584,-176.223,9.632,148.880
C07861=1144.893,373.633,-83.548,-176.226,9.628,148.879
C07862=1144.897,373.386,-83.511,-176.228,9.623,148.879
C07863=1144.901,373.138,-83.476,-176.231,9.619,148.878
C07864=1144.905,372.891,-83.439,-176.233,9.615,148.878
C07865=1144.909,372.643,-83.403,-176.236,9.611,148.878
C07866=1144.912,372.396,-83.367,-176.238,9.607,148.877
C07867=1144.916,372.149,-83.331,-176.241,9.602,148.877
C07868=1144.920,371.902,-83.295,-176.243,9.598,148.876
C07869=1144.924,371.654,-83.259,-176.246,9.594,148.876
C07870=1144.927,371.407,-83.222,-176.249,9.590,148.876
C07871=1144.932,371.159,-83.186,-176.250,9.586,148.875
C07872=1144.935,370.912,-83.150,-176.253,9.582,148.875
C07873=1144.940,370.665,-83.114,-176.255,9.577,148.874
C07874=1144.943,370.417,-83.078,-176.258,9.573,148.874
C07875=1144.947,370.170,-83.042,-176.261,9.569,148.874
C07876=1144.951,369.922,-83.006,-176.263,9.564,148.873
C07877=1144.955,369.675,-82.970,-176.266,9.560,148.873
C07878=1144.958,369.428,-82.934,-176.269,9.556,148.872
C07879=1144.962,369.180,-82.898,-176.271,9.552,148.872
C07880=1144.966,368.933,-82.862,-176.274,9.548,148.872
C07881=1144.969,368.686,-82.826,-176.276,9.544,148.871
C07882=1144.974,368.438,-82.790,-176.279,9.539,148.871
C07883=1144.977,368.190,-82.754,-176.282,9.535,148.870
C07884=1144.981,367.943,-82.719,-176.284,9.531,148.870
C07885=1144.986,367.695,-82.683,-176.287,9.527,148.870
C07886=1144.990,367.449,-82.647,-176.289,9.523,148.869
C07887=1144.993,367.202,-82.611,-176.292,9.518,148.869
C07888=1144.998,366.954,-82.575,-176.295,9.514,148.869
C07889=1145.001,366.706,-82.539,-176.297,9.510,148.868
C07890=1145.005,366.459,-82.504,-176.300,9.506,148.868
C07891=1145.009,366.211,-82.468,-176.302,9.502,148.867
C07892=1145.013,365.963,-82.432,-176.305,9.498,148.867
C07893=1145.017,365.717,-82.396,-176.308,9.494,148.867
C07894=1145.021,365.433,-82.355,-176.311,9.489,148.866
C07895=1145.025,365.149,-82.315,-176.314,9.484,148.866
C07896=1145.030,364.866,-82.274,-176.317,9.479,148.866
C07897=1145.034,364.582,-82.234,-176.320,9.475,148.865
C07898=1145.038,364.335,-82.198,-176.322,9.471,148.865
C07899=1145.042,364.088,-82.163,-176.325,9.467,148.864
C07900=1145.046,363.841,-82.127,-176.328,9.462,148.864
C07901=1145.050,363.593,-82.091,-176.331,9.458,148.864
C07902=1145.054,363.345,-82.056,-176.333,9.454,148.863
C07903=1145.058,363.098,-82.020,-176.335,9.450,148.863
C07904=1145.061,362.850,-81.985,-176.338,9.446,148.862
C07905=1145.066,362.603,-81.949,-176.341,9.442,148.862
C07906=1145.069,362.356,-81.914,-176.343,9.438,148.862
C07907=1145.073,362.108,-81.878,-176.346,9.433,148.861
C07908=1145.077,361.860,-81.843,-176.348,9.430,148.861
C07909=1145.081,361.614,-81.808,-176.351,9.426,148.861
C07910=1145.085,361.366,-81.773,-176.354,9.422,148.861
C07911=1145.088,361.119,-81.737,-176.356,9.417,148.860
C07912=1145.092,360.871,-81.702,-176.359,9.414,148.860
C07913=1145.097,360.624,-81.667,-176.361,9.410,148.859
C07914=1145.100,360.376,-81.632,-176.364,9.406,148.859
C07915=1145.104,360.129,-81.596,-176.367,9.401,148.859
C07916=1145.108,359.881,-81.560,-176.369,9.398,148.858
C07917=1145.112,359.634,-81.526,-176.372,9.394,148.858
C07918=1145.116,359.386,-81.490,-176.374,9.389,148.858
C07919=1145.120,359.139,-81.455,-176.377,9.385,148.857
C07920=1145.124,358.891,-81.420,-176.379,9.382,148.857
C07921=1145.128,358.644,-81.385,-176.382,9.377,148.857
C07922=1145.131,358.396,-81.349,-176.385,9.373,148.856
C07923=1145.135,358.148,-81.315,-176.387,9.370,148.856
C07924=1145.140,357.901,-81.279,-176.390,9.366,148.856
C07925=1145.144,357.653,-81.245,-176.392,9.361,148.855
C07926=1145.147,357.406,-81.209,-176.394,9.358,148.855
C07927=1145.152,357.159,-81.174,-176.397,9.354,148.855
C07928=1145.155,356.911,-81.140,-176.400,9.350,148.854
C07929=1145.159,356.664,-81.104,-176.402,9.346,148.854
C07930=1145.163,356.416,-81.070,-176.405,9.342,148.854
C07931=1145.167,356.169,-81.034,-176.407,9.338,148.853
C07932=1145.171,355.921,-81.000,-176.409,9.334,148.853
C07933=1145.175,355.674,-80.964,-176.412,9.330,148.853
C07934=1145.179,355.426,-80.929,-176.415,9.326,148.852
C07935=1145.183,355.179,-80.895,-176.417,9.322,148.852
C07936=1145.186,354.931,-80.860,-176.420,9.318,148.852
C07937=1145.191,354.684,-80.825,-176.422,9.314,148.851
C07938=1145.195,354.436,-80.790,-176.424,9.310,148.851
C07939=1145.199,354.188,-80.755,-176.427,9.306,148.850
C07940=1145.202,353.941,-80.721,-176.430,9.302,148.850
C07941=1145.206,353.693,-80.685,-176.432,9.298,148.850
C07942=1145.211,353.446,-80.651,-176.435,9.294,148.850
C07943=1145.215,353.198,-80.616,-176.438,9.290,148.849
C07944=1145.218,352.951,-80.582,-176.440,9.287,148.849
C07945=1145.222,352.703,-80.547,-176.442,9.283,148.849
C07946=1145.226,352.455,-80.512,-176.444,9.279,148.848
C07947=1145.231,352.208,-80.477,-176.447,9.275,148.848
C07948=1145.234,351.961,-80.442,-176.450,9.271,148.847
C07949=1145.238,351.713,-80.408,-176.452,9.267,148.847
C07950=1145.242,351.465,-80.373,-176.455,9.263,148.847
C07951=1145.246,351.218,-80.339,-176.458,9.259,148.847
C07952=1145.250,350.970,-80.304,-176.460,9.256,148.846
C07953=1145.254,350.723,-80.269,-176.462,9.251,148.846
C07954=1145.257,350.475,-80.235,-176.465,9.248,148.846
C07955=1145.262,350.228,-80.201,-176.467,9.243,148.845
C07956=1145.266,349.980,-80.166,-176.470,9.239,148.845
C07957=1145.270,349.733,-80.132,-176.472,9.236,148.845
C07958=1145.274,349.484,-80.097,-176.475,9.232,148.844
C07959=1145.278,349.237,-80.063,-176.477,9.228,148.844
C07960=1145.282,348.989,-80.028,-176.480,9.224,148.844
C07961=1145.286,348.742,-79.994,-176.483,9.220,148.843
C07962=1145.289,348.494,-79.960,-176.485,9.217,148.843
C07963=1145.294,348.246,-79.925,-176.487,9.212,148.843
C07964=1145.298,347.999,-79.891,-176.490,9.208,148.843
C07965=1145.302,347.751,-79.856,-176.493,9.205,148.842
C07966=1145.306,347.504,-79.823,-176.495,9.201,148.842
C07967=1145.310,347.256,-79.788,-176.498,9.197,148.842
C07968=1145.314,347.009,-79.753,-176.500,9.193,148.841
C07969=1145.317,346.761,-79.719,-176.502,9.190,148.841
C07970=1145.322,346.513,-79.685,-176.505,9.186,148.841
C07971=1145.326,346.266,-79.651,-176.508,9.181,148.840
C07972=1145.330,346.018,-79.616,-176.510,9.178,148.840
C07973=1145.334,345.771,-79.582,-176.513,9.174,148.840
C07974=1145.337,345.523,-79.547,-176.515,9.170,148.839
C07975=1145.342,345.275,-79.514,-176.518,9.166,148.839
C07976=1145.345,345.028,-79.480,-176.521,9.162,148.839
C07977=1145.349,344.780,-79.445,-176.523,9.159,148.839
C07978=1145.353,344.533,-79.411,-176.526,9.154,148.838
C07979=1145.358,344.285,-79.377,-176.528,9.151,148.838
C07980=1145.361,344.037,-79.343,-176.530,9.147,148.838
C07981=1145.366,343.790,-79.309,-176.533,9.144,148.837
C07982=1145.370,343.542,-79.275,-176.536,9.139,148.837
C07983=1145.373,343.295,-79.241,-176.538,9.135,148.837
C07984=1145.378,343.047,-79.207,-176.540,9.132,148.837
C07985=1145.382,342.800,-79.173,-176.543,9.128,148.836
C07986=1145.386,342.551,-79.138,-176.546,9.124,148.836
C07987=1145.390,342.304,-79.105,-176.548,9.120,148.836
C07988=1145.394,342.057,-79.071,-176.551,9.117,148.835
C07989=1145.398,341.808,-79.037,-176.553,9.113,148.835
C07990=1145.402,341.561,-79.003,-176.556,9.108,148.835
C07991=1145.406,341.314,-78.970,-176.558,9.105,148.835
C07992=1145.410,341.066,-78.936,-176.561,9.101,148.834
C07993=1145.414,340.818,-78.902,-176.564,9.098,148.834
C07994=1145.418,340.570,-78.868,-176.566,9.093,148.834
C07995=1145.422,340.323,-78.834,-176.568,9.090,148.833
C07996=1145.426,340.074,-78.800,-176.571,9.086,148.833
C07997=1145.430,339.827,-78.767,-176.574,9.083,148.833
C07998=1145.435,339.546,-78.728,-176.577,9.077,148.832
C07999=1145.439,339.267,-78.691,-176.580,9.073,148.832
C08000=1145.444,338.986,-78.652,-176.583,9.069,148.832
C08001=1145.449,338.706,-78.614,-176.585,9.065,148.832
C08002=1145.453,338.458,-78.580,-176.588,9.061,148.831
C08003=1145.456,338.210,-78.546,-176.590,9.058,148.831
C08004=1145.460,337.962,-78.513,-176.593,9.053,148.831
C08005=1145.464,337.715,-78.480,-176.595,9.050,148.831
C08006=1145.469,337.467,-78.445,-176.598,9.046,148.830
C08007=1145.473,337.220,-78.412,-176.600,9.043,148.830
C08008=1145.476,336.972,-78.378,-176.603,9.038,148.830
C08009=1145.480,336.724,-78.345,-176.606,9.035,148.830
C08010=1145.484,336.476,-78.312,-176.608,9.031,148.829
C08011=1145.489,336.229,-78.279,-176.610,9.028,148.829
C08012=1145.492,335.981,-78.245,-176.613,9.023,148.829
C08013=1145.496,335.733,-78.211,-176.616,9.020,148.828
C08014=1145.501,335.485,-78.177,-176.619,9.016,148.828
C08015=1145.505,335.238,-78.143,-176.621,9.013,148.828
C08016=1145.509,334.990,-78.110,-176.623,9.008,148.828
C08017=1145.513,334.742,-78.077,-176.626,9.005,148.827
C08018=1145.517,334.495,-78.044,-176.629,9.001,148.827
C08019=1145.521,334.246,-78.011,-176.631,8.998,148.827
C08020=1145.525,333.998,-77.977,-176.634,8.994,148.827
C08021=1145.529,333.751,-77.943,-176.636,8.990,148.826
C08022=1145.533,333.504,-77.910,-176.639,8.986,148.826
C08023=1145.537,333.256,-77.877,-176.641,8.983,148.826
C08024=1145.541,333.008,-77.844,-176.644,8.979,148.826
C08025=1145.545,332.760,-77.811,-176.646,8.975,148.825
C08026=1145.549,332.513,-77.778,-176.649,8.971,148.825
C08027=1145.553,332.265,-77.745,-176.651,8.968,148.825
C08028=1145.557,332.017,-77.711,-176.654,8.964,148.825
C08029=1145.561,331.769,-77.678,-176.656,8.960,148.824
C08030=1145.565,331.521,-77.645,-176.659,8.956,148.824
C08031=1145.569,331.273,-77.612,-176.662,8.953,148.824
C08032=1145.574,331.026,-77.578,-176.664,8.949,148.824
C08033=1145.578,330.778,-77.545,-176.667,8.946,148.824
C08034=1145.582,330.530,-77.512,-176.670,8.942,148.823
C08035=1145.586,330.282,-77.479,-176.672,8.938,148.823
C08036=1145.589,330.035,-77.446,-176.675,8.934,148.823
C08037=1145.593,329.787,-77.413,-176.677,8.931,148.822
C08038=1145.598,329.540,-77.380,-176.680,8.927,148.822
C08039=1145.602,329.292,-77.347,-176.682,8.923,148.822
C08040=1145.606,329.044,-77.314,-176.685,8.919,148.822
C08041=1145.610,328.796,-77.281,-176.687,8.916,148.822
C08042=1145.614,328.548,-77.248,-176.690,8.912,148.821
C08043=1145.619,328.300,-77.215,-176.693,8.909,148.821
C08044=1145.622,328.053,-77.182,-176.696,8.905,148.821
C08045=1145.626,327.805,-77.149,-176.698,8.901,148.821
C08046=1145.630,327.557,-77.116,-176.700,8.898,148.821
C08047=1145.635,327.309,-77.084,-176.703,8.894,148.820
C08048=1145.639,327.061,-77.051,-176.705,8.891,148.820
C08049=1145.642,326.814,-77.018,-176.708,8.887,148.820
C08050=1145.646,326.566,-76.985,-176.710,8.883,148.819
C08051=1145.651,326.318,-76.952,-176.713,8.879,148.819
C08052=1145.655,326.070,-76.919,-176.715,8.876,148.819
C08053=1145.658,325.823,-76.887,-176.718,8.872,148.819
C08054=1145.663,325.574,-76.854,-176.721,8.868,148.819
C08055=1145.667,325.327,-76.821,-176.724,8.864,148.818
C08056=1145.671,325.079,-76.788,-176.726,8.861,148.818
C08057=1145.675,324.831,-76.756,-176.728,8.858,148.818
C08058=1145.679,324.583,-76.723,-176.731,8.854,148.818
C08059=1145.683,324.335,-76.690,-176.734,8.850,148.818
C08060=1145.687,324.087,-76.658,-176.736,8.846,148.817
C08061=1145.692,323.840,-76.625,-176.739,8.843,148.817
C08062=1145.696,323.592,-76.593,-176.742,8.839,148.817
C08063=1145.699,323.345,-76.560,-176.744,8.836,148.817
C08064=1145.704,323.096,-76.528,-176.746,8.832,148.817
C08065=1145.708,322.848,-76.495,-176.749,8.828,148.816
C08066=1145.712,322.600,-76.463,-176.752,8.825,148.816
C08067=1145.716,322.353,-76.430,-176.755,8.821,148.816
C08068=1145.719,322.105,-76.398,-176.757,8.818,148.816
C08069=1145.724,321.857,-76.365,-176.760,8.814,148.815
C08070=1145.729,321.609,-76.332,-176.762,8.810,148.815
C08071=1145.732,321.362,-76.300,-176.764,8.807,148.815
C08072=1145.737,321.114,-76.267,-176.767,8.803,148.815
C08073=1145.740,320.865,-76.236,-176.770,8.800,148.815
C08074=1145.744,320.618,-76.202,-176.773,8.796,148.815
C08075=1145.748,320.370,-76.171,-176.775,8.793,148.814
C08076=1145.752,320.122,-76.137,-176.778,8.789,148.814
C08077=1145.757,319.875,-76.106,-176.781,8.785,148.814
C08078=1145.761,319.626,-76.074,-176.783,8.782,148.814
C08079=1145.764,319.379,-76.041,-176.786,8.778,148.814
C08080=1145.769,319.131,-76.009,-176.788,8.775,148.813
C08081=1145.773,318.883,-75.977,-176.791,8.771,148.813
C08082=1145.778,318.635,-75.945,-176.793,8.767,148.813
C08083=1145.781,318.387,-75.912,-176.796,8.764,148.813
C08084=1145.785,318.139,-75.880,-176.799,8.760,148.813
C08085=1145.789,317.891,-75.848,-176.801,8.757,148.812
C08086=1145.794,317.643,-75.815,-176.803,8.754,148.812
C08087=1145.798,317.396,-75.783,-176.806,8.749,148.812
C08088=1145.802,317.148,-75.751,-176.809,8.747,148.812
C08089=1145.806,316.900,-75.719,-176.812,8.742,148.812
C08090=1145.809,316.652,-75.687,-176.814,8.739,148.812
C08091=1145.814,316.404,-75.655,-176.817,8.736,148.811
C08092=1145.818,316.156,-75.623,-176.819,8.732,148.811
C08093=1145.823,315.908,-75.591,-176.822,8.729,148.811
C08094=1145.826,315.659,-75.559,-176.825,8.724,148.811
C08095=1145.830,315.413,-75.527,-176.827,8.721,148.811
C08096=1145.835,315.164,-75.494,-176.830,8.718,148.811
C08097=1145.838,314.916,-75.462,-176.833,8.714,148.810
C08098=1145.843,314.669,-75.431,-176.835,8.711,148.810
C08099=1145.847,314.421,-75.398,-176.837,8.708,148.810
C08100=1145.851,314.173,-75.367,-176.840,8.704,148.810
C08101=1145.855,313.925,-75.335,-176.843,8.700,148.810
C08102=1145.860,313.647,-75.298,-176.846,8.696,148.809
C08103=1145.865,313.369,-75.264,-176.849,8.692,148.809
C08104=1145.869,313.092,-75.228,-176.852,8.688,148.809
C08105=1145.874,312.814,-75.192,-176.855,8.684,148.809
C08106=1145.878,312.566,-75.160,-176.857,8.681,148.809
C08107=1145.882,312.318,-75.128,-176.859,8.678,148.809
C08108=1145.886,312.071,-75.097,-176.862,8.674,148.808
C08109=1145.890,311.822,-75.065,-176.865,8.671,148.808
C08110=1145.894,311.574,-75.033,-176.868,8.667,148.808
C08111=1145.899,311.326,-75.002,-176.870,8.663,148.808
C08112=1145.902,311.078,-74.970,-176.873,8.660,148.808
C08113=1145.906,310.830,-74.938,-176.876,8.656,148.808
C08114=1145.911,310.582,-74.906,-176.878,8.653,148.808
C08115=1145.915,310.334,-74.874,-176.881,8.650,148.807
C08116=1145.920,310.086,-74.844,-176.884,8.646,148.807
C08117=1145.923,309.838,-74.812,-176.886,8.642,148.807
C08118=1145.927,309.590,-74.780,-176.888,8.639,148.807
C08119=1145.932,309.343,-74.748,-176.892,8.635,148.807
C08120=1145.936,309.094,-74.717,-176.894,8.632,148.807
C08121=1145.940,308.847,-74.685,-176.896,8.629,148.806
C08122=1145.944,308.599,-74.653,-176.899,8.625,148.806
C08123=1145.949,308.351,-74.623,-176.902,8.622,148.806
C08124=1145.952,308.103,-74.591,-176.904,8.619,148.806
C08125=1145.957,307.855,-74.559,-176.907,8.615,148.806
C08126=1145.961,307.607,-74.528,-176.910,8.611,148.806
C08127=1145.964,307.359,-74.496,-176.912,8.608,148.806
C08128=1145.969,307.111,-74.465,-176.915,8.604,148.805
C08129=1145.973,306.862,-74.433,-176.918,8.601,148.805
C08130=1145.978,306.615,-74.402,-176.920,8.598,148.805
C08131=1145.982,306.366,-74.370,-176.923,8.594,148.805
C08132=1145.986,306.119,-74.339,-176.926,8.591,148.805
C08133=1145.990,305.870,-74.308,-176.928,8.587,148.805
C08134=1145.994,305.623,-74.276,-176.931,8.583,148.805
C08135=1145.998,305.374,-74.245,-176.934,8.580,148.805
C08136=1146.003,305.127,-74.214,-176.936,8.577,148.804
C08137=1146.007,304.878,-74.183,-176.938,8.574,148.804
C08138=1146.011,304.631,-74.151,-176.942,8.570,148.804
C08139=1146.015,304.382,-74.120,-176.944,8.567,148.804
C08140=1146.019,304.135,-74.089,-176.946,8.564,148.804
C08141=1146.024,303.887,-74.058,-176.949,8.560,148.804
C08142=1146.028,303.638,-74.027,-176.952,8.557,148.804
C08143=1146.032,303.391,-73.995,-176.954,8.553,148.803
C08144=1146.036,303.142,-73.964,-176.957,8.549,148.803
C08145=1146.040,302.895,-73.934,-176.960,8.546,148.803
C08146=1146.044,302.647,-73.902,-176.962,8.543,148.803
C08147=1146.048,302.399,-73.871,-176.965,8.540,148.803
C08148=1146.052,302.150,-73.840,-176.968,8.536,148.803
C08149=1146.057,301.903,-73.809,-176.970,8.533,148.803
C08150=1146.061,301.655,-73.778,-176.973,8.529,148.803
C08151=1146.065,301.406,-73.747,-176.976,8.526,148.803
C08152=1146.070,301.159,-73.715,-176.978,8.522,148.802
C08153=1146.074,300.910,-73.684,-176.981,8.519,148.802
C08154=1146.078,300.663,-73.654,-176.984,8.515,148.802
C08155=1146.082,300.415,-73.623,-176.986,8.512,148.802
C08156=1146.086,300.166,-73.592,-176.989,8.509,148.802
C08157=1146.091,299.919,-73.561,-176.991,8.506,148.802
C08158=1146.095,299.671,-73.530,-176.994,8.502,148.802
C08159=1146.098,299.422,-73.499,-176.997,8.499,148.802
C08160=1146.103,299.174,-73.469,-176.999,8.496,148.802
C08161=1146.107,298.926,-73.437,-177.002,8.492,148.801
C08162=1146.112,298.678,-73.407,-177.005,8.489,148.801
C08163=1146.116,298.430,-73.376,-177.007,8.485,148.801
C08164=1146.119,298.182,-73.345,-177.010,8.482,148.801
C08165=1146.124,297.934,-73.314,-177.013,8.478,148.801
C08166=1146.128,297.686,-73.283,-177.015,8.475,148.801
C08167=1146.132,297.438,-73.253,-177.018,8.472,148.801
C08168=1146.136,297.190,-73.222,-177.021,8.469,148.801
C08169=1146.141,296.942,-73.191,-177.023,8.465,148.800
C08170=1146.145,296.694,-73.161,-177.026,8.462,148.800
C08171=1146.149,296.446,-73.130,-177.029,8.459,148.800
C08172=1146.153,296.198,-73.099,-177.031,8.456,148.800
C08173=1146.157,295.950,-73.069,-177.034,8.452,148.800
C08174=1146.161,295.701,-73.038,-177.037,8.449,148.800
C08175=1146.166,295.453,-73.007,-177.039,8.445,148.800
C08176=1146.170,295.205,-72.977,-177.042,8.442,148.800
C08177=1146.174,294.956,-72.946,-177.045,8.438,148.800
C08178=1146.179,294.708,-72.916,-177.047,8.435,148.800
C08179=1146.183,294.461,-72.885,-177.050,8.432,148.800
C08180=1146.187,294.213,-72.855,-177.052,8.429,148.800
C08181=1146.191,293.964,-72.824,-177.056,8.425,148.800
C08182=1146.195,293.716,-72.793,-177.058,8.422,148.799
C08183=1146.199,293.469,-72.763,-177.061,8.419,148.799
C08184=1146.204,293.220,-72.733,-177.063,8.416,148.799
C08185=1146.208,292.972,-72.702,-177.066,8.412,148.799
C08186=1146.212,292.724,-72.672,-177.069,8.409,148.799
C08187=1146.216,292.476,-72.641,-177.071,8.405,148.799
C08188=1146.221,292.228,-72.612,-177.074,8.402,148.799
C08189=1146.225,291.980,-72.581,-177.076,8.399,148.799
C08190=1146.229,291.731,-72.550,-177.080,8.395,148.799
C08191=1146.233,291.483,-72.520,-177.082,8.392,148.799
C08192=1146.237,291.235,-72.490,-177.085,8.389,148.799
C08193=1146.242,290.987,-72.459,-177.087,8.386,148.798
C08194=1146.246,290.740,-72.429,-177.090,8.383,148.798
C08195=1146.250,290.490,-72.399,-177.093,8.379,148.798
C08196=1146.254,290.243,-72.369,-177.096,8.376,148.798
C08197=1146.258,289.995,-72.338,-177.098,8.373,148.798
C08198=1146.263,289.746,-72.308,-177.101,8.370,148.798
C08199=1146.267,289.499,-72.278,-177.104,8.366,148.798
C08200=1146.272,289.250,-72.248,-177.106,8.363,148.798
C08201=1146.275,289.003,-72.218,-177.109,8.359,148.798
C08202=1146.280,288.753,-72.188,-177.112,8.357,148.798
C08203=1146.284,288.506,-72.157,-177.114,8.353,148.798
C08204=1146.288,288.257,-72.128,-177.117,8.350,148.798
C08205=1146.292,288.009,-72.097,-177.120,8.346,148.798
C08206=1146.297,287.735,-72.064,-177.122,8.343,148.798
C08207=1146.301,287.459,-72.031,-177.126,8.340,148.798
C08208=1146.306,287.184,-71.998,-177.129,8.335,148.797
C08209=1146.311,286.907,-71.964,-177.131,8.333,148.797
C08210=1146.315,286.660,-71.934,-177.134,8.328,148.797
C08211=1146.319,286.411,-71.904,-177.137,8.326,148.797
C08212=1146.324,286.164,-71.874,-177.140,8.323,148.797
C08213=1146.328,285.915,-71.844,-177.142,8.319,148.797
C08214=1146.332,285.667,-71.815,-177.145,8.316,148.797
C08215=1146.337,285.419,-71.784,-177.148,8.312,148.797
C08216=1146.341,285.171,-71.754,-177.151,8.309,148.797
C08217=1146.345,284.922,-71.725,-177.153,8.306,148.797
C08218=1146.349,284.675,-71.695,-177.156,8.303,148.797
C08219=1146.354,284.426,-71.665,-177.158,8.300,148.797
C08220=1146.358,284.178,-71.635,-177.161,8.297,148.797
C08221=1146.362,283.930,-71.605,-177.164,8.293,148.797
C08222=1146.366,283.682,-71.576,-177.167,8.290,148.797
C08223=1146.371,283.434,-71.546,-177.169,8.287,148.797
C08224=1146.375,283.185,-71.516,-177.172,8.284,148.797
C08225=1146.379,282.938,-71.486,-177.174,8.281,148.797
C08226=1146.383,282.689,-71.457,-177.177,8.278,148.797
C08227=1146.388,282.441,-71.427,-177.180,8.274,148.796
C08228=1146.392,282.193,-71.398,-177.183,8.271,148.796
C08229=1146.397,281.944,-71.368,-177.186,8.268,148.796
C08230=1146.401,281.697,-71.337,-177.188,8.265,148.796
C08231=1146.405,281.448,-71.308,-177.191,8.262,148.796
C08232=1146.409,281.200,-71.279,-177.193,8.258,148.796
C08233=1146.413,280.952,-71.249,-177.196,8.255,148.796
C08234=1146.417,280.704,-71.220,-177.199,8.252,148.796
C08235=1146.421,280.455,-71.190,-177.202,8.248,148.796
C08236=1146.426,280.207,-71.160,-177.204,8.246,148.796
C08237=1146.431,279.958,-71.131,-177.207,8.243,148.796
C08238=1146.435,279.710,-71.101,-177.209,8.239,148.796
C08239=1146.439,279.462,-71.072,-177.212,8.236,148.796
C08240=1146.443,279.214,-71.042,-177.215,8.232,148.796
C08241=1146.447,278.965,-71.013,-177.218,8.229,148.796
C08242=1146.452,278.718,-70.984,-177.221,8.226,148.796
C08243=1146.456,278.469,-70.954,-177.223,8.223,148.796
C08244=1146.460,278.221,-70.925,-177.226,8.220,148.796
C08245=1146.465,277.973,-70.895,-177.229,8.217,148.796
C08246=1146.469,277.725,-70.866,-177.231,8.214,148.796
C08247=1146.473,277.476,-70.837,-177.234,8.210,148.796
C08248=1146.477,277.228,-70.807,-177.237,8.207,148.796
C08249=1146.481,276.980,-70.778,-177.239,8.204,148.796
C08250=1146.485,276.732,-70.748,-177.242,8.201,148.796
C08251=1146.490,276.484,-70.719,-177.245,8.198,148.796
C08252=1146.495,276.235,-70.690,-177.248,8.195,148.796
C08253=1146.499,275.987,-70.661,-177.250,8.192,148.796
C08254=1146.503,275.739,-70.631,-177.253,8.189,148.796
C08255=1146.507,275.490,-70.602,-177.256,8.185,148.796
C08256=1146.511,275.242,-70.573,-177.258,8.182,148.796
C08257=1146.515,274.994,-70.544,-177.261,8.179,148.796
C08258=1146.520,274.746,-70.515,-177.264,8.176,148.796
C08259=1146.524,274.498,-70.486,-177.266,8.173,148.796
C08260=1146.528,274.249,-70.456,-177.269,8.170,148.796
C08261=1146.533,274.001,-70.428,-177.272,8.167,148.796
C08262=1146.537,273.752,-70.398,-177.275,8.164,148.796
C08263=1146.542,273.505,-70.369,-177.278,8.160,148.795
C08264=1146.545,273.257,-70.340,-177.280,8.157,148.796
C08265=1146.550,273.008,-70.312,-177.283,8.154,148.796
C08266=1146.554,272.760,-70.282,-177.286,8.151,148.795
C08267=1146.558,272.511,-70.253,-177.288,8.148,148.795
C08268=1146.563,272.263,-70.224,-177.291,8.145,148.796
C08269=1146.567,272.015,-70.195,-177.294,8.142,148.796
C08270=1146.571,271.766,-70.167,-177.296,8.139,148.795
C08271=1146.575,271.518,-70.137,-177.299,8.136,148.795
C08272=1146.580,271.270,-70.109,-177.302,8.133,148.796
C08273=1146.585,271.022,-70.079,-177.305,8.129,148.796
C08274=1146.588,270.774,-70.051,-177.307,8.126,148.795
C08275=1146.593,270.525,-70.022,-177.310,8.123,148.795
C08276=1146.597,270.277,-69.993,-177.313,8.120,148.795
C08277=1146.602,270.028,-69.964,-177.316,8.117,148.796
C08278=1146.605,269.780,-69.935,-177.318,8.114,148.795
C08279=1146.610,269.532,-69.907,-177.321,8.111,148.795
C08280=1146.615,269.284,-69.877,-177.324,8.108,148.796
C08281=1146.618,269.035,-69.849,-177.326,8.105,148.796
C08282=1146.623,268.786,-69.820,-177.329,8.102,148.796
C08283=1146.628,268.539,-69.791,-177.332,8.099,148.795
C08284=1146.631,268.290,-69.763,-177.334,8.096,148.796
C08285=1146.635,268.042,-69.734,-177.338,8.092,148.796
C08286=1146.641,267.794,-69.705,-177.340,8.089,148.796
C08287=1146.644,267.545,-69.677,-177.343,8.086,148.795
C08288=1146.648,267.297,-69.648,-177.346,8.083,148.796
C08289=1146.654,267.049,-69.619,-177.348,8.080,148.796
C08290=1146.657,266.800,-69.591,-177.351,8.077,148.796
C08291=1146.662,266.553,-69.562,-177.354,8.074,148.796
C08292=1146.667,266.304,-69.533,-177.356,8.071,148.796
C08293=1146.670,266.055,-69.505,-177.359,8.068,148.796
C08294=1146.675,265.808,-69.476,-177.362,8.065,148.796
C08295=1146.679,265.559,-69.448,-177.365,8.062,148.796
C08296=1146.683,265.310,-69.419,-177.367,8.059,148.796
C08297=1146.688,265.062,-69.392,-177.370,8.056,148.796
C08298=1146.692,264.813,-69.363,-177.373,8.053,148.796
C08299=1146.696,264.566,-69.334,-177.375,8.050,148.796
C08300=1146.701,264.317,-69.306,-177.378,8.047,148.796
C08301=1146.705,264.068,-69.277,-177.381,8.043,148.796
C08302=1146.710,263.820,-69.249,-177.384,8.041,148.796
C08303=1146.714,263.572,-69.220,-177.387,8.038,148.796
C08304=1146.718,263.324,-69.193,-177.389,8.034,148.796
C08305=1146.723,263.075,-69.163,-177.392,8.031,148.796
C08306=1146.727,262.828,-69.135,-177.395,8.029,148.796
C08307=1146.731,262.579,-69.107,-177.398,8.026,148.796
C08308=1146.735,262.330,-69.078,-177.400,8.023,148.796
C08309=1146.740,262.082,-69.051,-177.403,8.020,148.796
C08310=1146.745,261.809,-69.019,-177.406,8.017,148.796
C08311=1146.750,261.535,-68.989,-177.409,8.013,148.796
C08312=1146.753,261.262,-68.957,-177.412,8.010,148.796
C08313=1146.759,260.988,-68.926,-177.415,8.006,148.796
C08314=1146.763,260.740,-68.898,-177.418,8.003,148.796
C08315=1146.768,260.491,-68.869,-177.421,8.000,148.796
C08316=1146.772,260.244,-68.841,-177.423,7.997,148.796
C08317=1146.776,259.995,-68.813,-177.426,7.994,148.796
C08318=1146.781,259.746,-68.786,-177.429,7.991,148.796
C08319=1146.785,259.498,-68.757,-177.432,7.988,148.796
C08320=1146.789,259.250,-68.730,-177.435,7.986,148.796
C08321=1146.794,259.001,-68.701,-177.437,7.982,148.796
C08322=1146.798,258.753,-68.673,-177.440,7.979,148.796
C08323=1146.802,258.504,-68.645,-177.442,7.976,148.796
C08324=1146.807,258.256,-68.617,-177.445,7.973,148.797
C08325=1146.811,258.008,-68.588,-177.448,7.971,148.797
C08326=1146.815,257.759,-68.561,-177.451,7.968,148.797
C08327=1146.820,257.511,-68.533,-177.454,7.965,148.797
C08328=1146.824,257.262,-68.505,-177.456,7.962,148.797
C08329=1146.828,257.014,-68.477,-177.459,7.959,148.797
C08330=1146.832,256.766,-68.449,-177.462,7.956,148.797
C08331=1146.838,256.517,-68.421,-177.464,7.953,148.797
C08332=1146.841,256.268,-68.393,-177.467,7.950,148.797
C08333=1146.846,256.021,-68.365,-177.470,7.947,148.797
C08334=1146.850,255.773,-68.338,-177.473,7.944,148.797
C08335=1146.855,255.523,-68.310,-177.475,7.941,148.797
C08336=1146.859,255.275,-68.282,-177.478,7.938,148.797
C08337=1146.863,255.027,-68.254,-177.481,7.935,148.797
C08338=1146.868,254.778,-68.227,-177.484,7.932,148.797
C08339=1146.872,254.530,-68.199,-177.487,7.929,148.797
C08340=1146.876,254.282,-68.171,-177.489,7.926,148.797
C08341=1146.881,254.033,-68.143,-177.492,7.923,148.797
C08342=1146.885,253.785,-68.115,-177.495,7.920,148.797
C08343=1146.890,253.536,-68.088,-177.498,7.917,148.798
C08344=1146.894,253.288,-68.060,-177.500,7.915,148.798
C08345=1146.898,253.040,-68.032,-177.503,7.912,148.798
C08346=1146.902,252.791,-68.005,-177.506,7.909,148.798
C08347=1146.907,252.543,-67.977,-177.508,7.905,148.798
C08348=1146.911,252.294,-67.949,-177.511,7.902,148.798
C08349=1146.916,252.046,-67.921,-177.514,7.900,148.798
C08350=1146.920,251.797,-67.894,-177.517,7.897,148.798
C08351=1146.924,251.549,-67.866,-177.520,7.894,148.798
C08352=1146.929,251.300,-67.839,-177.522,7.891,148.798
C08353=1146.933,251.052,-67.811,-177.525,7.889,148.798
C08354=1146.938,250.804,-67.784,-177.527,7.886,148.798
C08355=1146.942,250.555,-67.756,-177.530,7.883,148.798
C08356=1146.946,250.307,-67.729,-177.533,7.880,148.798
C08357=1146.951,250.058,-67.702,-177.536,7.877,148.798
C08358=1146.955,249.810,-67.674,-177.538,7.874,148.798
C08359=1146.959,249.561,-67.647,-177.541,7.871,148.798
C08360=1146.964,249.313,-67.620,-177.544,7.868,148.799
C08361=1146.968,249.065,-67.592,-177.547,7.865,148.799
C08362=1146.972,248.816,-67.564,-177.550,7.862,148.799
C08363=1146.977,248.567,-67.537,-177.552,7.859,148.799
C08364=1146.981,248.319,-67.510,-177.555,7.856,148.799
C08365=1146.986,248.071,-67.483,-177.558,7.854,148.799
C08366=1146.990,247.822,-67.455,-177.561,7.851,148.799
C08367=1146.994,247.574,-67.427,-177.564,7.848,148.799
C08368=1146.999,247.325,-67.400,-177.566,7.845,148.799
C08369=1147.004,247.077,-67.373,-177.569,7.842,148.799
C08370=1147.007,246.828,-67.346,-177.572,7.839,148.799
C08371=1147.011,246.580,-67.319,-177.575,7.836,148.799
C08372=1147.016,246.331,-67.292,-177.577,7.834,148.799
C08373=1147.021,246.083,-67.264,-177.580,7.831,148.800
C08374=1147.025,245.834,-67.237,-177.582,7.828,148.800
C08375=1147.030,245.586,-67.210,-177.585,7.825,148.800
C08376=1147.034,245.337,-67.183,-177.588,7.822,148.800
C08377=1147.038,245.089,-67.155,-177.591,7.819,148.800
C08378=1147.042,244.841,-67.129,-177.594,7.816,148.800
C08379=1147.047,244.592,-67.102,-177.596,7.813,148.800
C08380=1147.052,244.344,-67.075,-177.599,7.810,148.800
C08381=1147.056,244.095,-67.048,-177.602,7.808,148.800
C08382=1147.060,243.846,-67.020,-177.605,7.805,148.800
C08383=1147.064,243.598,-66.994,-177.608,7.802,148.800
C08384=1147.069,243.349,-66.967,-177.611,7.799,148.801
C08385=1147.074,243.101,-66.939,-177.613,7.797,148.801
C08386=1147.078,242.852,-66.912,-177.616,7.794,148.801
C08387=1147.083,242.604,-66.885,-177.619,7.791,148.801
C08388=1147.087,242.356,-66.859,-177.621,7.788,148.801
C08389=1147.091,242.106,-66.831,-177.624,7.785,148.801
C08390=1147.096,241.858,-66.804,-177.627,7.782,148.801
C08391=1147.099,241.610,-66.778,-177.630,7.779,148.801
C08392=1147.104,241.361,-66.751,-177.633,7.777,148.801
C08393=1147.109,241.113,-66.724,-177.635,7.774,148.801
C08394=1147.113,240.864,-66.697,-177.638,7.771,148.801
C08395=1147.117,240.616,-66.670,-177.641,7.768,148.801
C08396=1147.122,240.368,-66.643,-177.643,7.766,148.802
C08397=1147.127,240.119,-66.616,-177.646,7.763,148.802
C08398=1147.131,239.870,-66.590,-177.649,7.760,148.802
C08399=1147.136,239.622,-66.563,-177.652,7.757,148.802
C08400=1147.140,239.373,-66.536,-177.655,7.754,148.802
C08401=1147.144,239.125,-66.510,-177.657,7.751,148.802
C08402=1147.149,238.877,-66.483,-177.660,7.748,148.802
C08403=1147.152,238.627,-66.457,-177.663,7.745,148.802
C08404=1147.157,238.379,-66.430,-177.665,7.743,148.802
C08405=1147.162,238.130,-66.403,-177.668,7.740,148.802
C08406=1147.166,237.882,-66.376,-177.671,7.738,148.803
C08407=1147.171,237.633,-66.350,-177.674,7.735,148.803
C08408=1147.175,237.385,-66.323,-177.677,7.732,148.803
C08409=1147.179,237.136,-66.296,-177.680,7.729,148.803
C08410=1147.184,236.888,-66.269,-177.682,7.726,148.803
C08411=1147.188,236.639,-66.243,-177.685,7.723,148.803
C08412=1147.193,236.390,-66.216,-177.687,7.721,148.803
C08413=1147.197,236.142,-66.190,-177.690,7.718,148.803
C08414=1147.202,235.870,-66.161,-177.694,7.714,148.803
C08415=1147.206,235.599,-66.132,-177.697,7.712,148.804
C08416=1147.212,235.327,-66.103,-177.700,7.709,148.804
C08417=1147.217,235.055,-66.074,-177.702,7.706,148.804
C08418=1147.221,234.807,-66.048,-177.705,7.703,148.804
C08419=1147.226,234.558,-66.022,-177.708,7.700,148.804
C08420=1147.230,234.309,-65.995,-177.711,7.697,148.804
C08421=1147.235,234.060,-65.969,-177.714,7.695,148.804
C08422=1147.239,233.812,-65.942,-177.716,7.693,148.805
C08423=1147.243,233.564,-65.915,-177.719,7.690,148.805
C08424=1147.248,233.315,-65.890,-177.722,7.687,148.805
C08425=1147.252,233.067,-65.863,-177.725,7.684,148.805
C08426=1147.256,232.817,-65.837,-177.727,7.681,148.805
C08427=1147.261,232.569,-65.811,-177.730,7.678,148.805
C08428=1147.265,232.320,-65.784,-177.733,7.675,148.805
C08429=1147.270,232.072,-65.759,-177.736,7.673,148.805
C08430=1147.274,231.824,-65.732,-177.738,7.670,148.805
C08431=1147.279,231.575,-65.706,-177.741,7.667,148.806
C08432=1147.283,231.327,-65.679,-177.744,7.665,148.806
C08433=1147.287,231.078,-65.654,-177.747,7.662,148.806
C08434=1147.292,230.829,-65.627,-177.750,7.660,148.806
C08435=1147.296,230.580,-65.601,-177.752,7.657,148.806
C08436=1147.301,230.331,-65.574,-177.755,7.654,148.806
C08437=1147.306,230.083,-65.549,-177.758,7.651,148.806
C08438=1147.310,229.835,-65.523,-177.761,7.648,148.806
C08439=1147.314,229.586,-65.497,-177.764,7.646,148.807
C08440=1147.319,229.337,-65.470,-177.766,7.643,148.807
C08441=1147.323,229.089,-65.444,-177.769,7.641,148.807
C08442=1147.327,228.840,-65.418,-177.772,7.638,148.807
C08443=1147.333,228.592,-65.392,-177.775,7.635,148.807
C08444=1147.337,228.343,-65.366,-177.777,7.632,148.807
C08445=1147.341,228.095,-65.340,-177.780,7.630,148.807
C08446=1147.345,227.846,-65.314,-177.783,7.627,148.808
C08447=1147.350,227.597,-65.288,-177.786,7.624,148.808
C08448=1147.355,227.349,-65.263,-177.788,7.621,148.808
C08449=1147.359,227.100,-65.237,-177.791,7.618,148.808
C08450=1147.363,226.852,-65.210,-177.794,7.617,148.808
C08451=1147.367,226.603,-65.185,-177.797,7.614,148.808
C08452=1147.373,226.355,-65.159,-177.799,7.611,148.808
C08453=1147.377,226.106,-65.133,-177.802,7.608,148.808
C08454=1147.381,225.857,-65.107,-177.805,7.605,148.809
C08455=1147.385,225.608,-65.081,-177.808,7.603,148.809
C08456=1147.390,225.359,-65.056,-177.810,7.600,148.809
C08457=1147.395,225.111,-65.030,-177.813,7.597,148.809
C08458=1147.399,224.862,-65.004,-177.816,7.594,148.809
C08459=1147.404,224.613,-64.978,-177.819,7.592,148.809
C08460=1147.409,224.365,-64.953,-177.822,7.590,148.810
C08461=1147.413,224.116,-64.927,-177.824,7.587,148.810
C08462=1147.417,223.868,-64.901,-177.827,7.584,148.810
C08463=1147.421,223.619,-64.875,-177.830,7.581,148.810
C08464=1147.426,223.371,-64.850,-177.833,7.579,148.810
C08465=1147.430,223.122,-64.824,-177.835,7.576,148.810
C08466=1147.434,222.873,-64.799,-177.838,7.573,148.810
C08467=1147.439,222.625,-64.773,-177.841,7.571,148.811
C08468=1147.444,222.376,-64.747,-177.844,7.569,148.811
C08469=1147.448,222.127,-64.721,-177.846,7.566,148.811
C08470=1147.453,221.879,-64.696,-177.849,7.563,148.811
C08471=1147.458,221.630,-64.670,-177.852,7.560,148.811
C08472=1147.462,221.381,-64.644,-177.855,7.558,148.811
C08473=1147.467,221.133,-64.619,-177.858,7.555,148.811
C08474=1147.471,220.884,-64.593,-177.860,7.552,148.812
C08475=1147.475,220.635,-64.568,-177.864,7.550,148.812
C08476=1147.480,220.387,-64.543,-177.866,7.548,148.812
C08477=1147.484,220.138,-64.517,-177.869,7.545,148.812
C08478=1147.489,219.889,-64.491,-177.871,7.542,148.812
C08479=1147.493,219.641,-64.466,-177.875,7.539,148.812
C08480=1147.497,219.392,-64.441,-177.877,7.537,148.813
C08481=1147.501,219.143,-64.416,-177.880,7.534,148.813
C08482=1147.506,218.895,-64.390,-177.883,7.532,148.813
C08483=1147.511,218.646,-64.364,-177.886,7.529,148.813
C08484=1147.516,218.398,-64.340,-177.888,7.527,148.813
C08485=1147.520,218.149,-64.314,-177.891,7.524,148.813
C08486=1147.524,217.900,-64.288,-177.894,7.521,148.814
C08487=1147.529,217.651,-64.264,-177.897,7.518,148.814
C08488=1147.533,217.402,-64.238,-177.899,7.516,148.814
C08489=1147.538,217.154,-64.212,-177.902,7.514,148.814
C08490=1147.542,216.905,-64.188,-177.905,7.511,148.814
C08491=1147.547,216.657,-64.163,-177.907,7.509,148.814
C08492=1147.551,216.408,-64.137,-177.910,7.506,148.814
C08493=1147.556,216.159,-64.112,-177.913,7.503,148.815
C08494=1147.560,215.911,-64.086,-177.916,7.500,148.815
C08495=1147.565,215.661,-64.061,-177.918,7.498,148.815
C08496=1147.569,215.414,-64.037,-177.922,7.495,148.815
C08497=1147.573,215.165,-64.011,-177.924,7.493,148.815
C08498=1147.578,214.916,-63.986,-177.927,7.490,148.816
C08499=1147.583,214.667,-63.960,-177.930,7.488,148.816
C08500=1147.588,214.419,-63.936,-177.933,7.485,148.816
C08501=1147.591,214.170,-63.911,-177.935,7.483,148.816
C08502=1147.596,213.921,-63.886,-177.938,7.480,148.816
C08503=1147.601,213.673,-63.860,-177.941,7.477,148.816
C08504=1147.606,213.424,-63.836,-177.944,7.474,148.817
C08505=1147.610,213.175,-63.811,-177.946,7.473,148.817
C08506=1147.614,212.927,-63.786,-177.949,7.470,148.817
C08507=1147.619,212.677,-63.761,-177.952,7.467,148.817
C08508=1147.624,212.429,-63.735,-177.955,7.465,148.817
C08509=1147.628,212.180,-63.711,-177.957,7.462,148.818
C08510=1147.632,211.932,-63.685,-177.960,7.459,148.818
C08511=1147.637,211.682,-63.660,-177.963,7.458,148.818
C08512=1147.641,211.434,-63.636,-177.966,7.455,148.818
C08513=1147.646,211.186,-63.611,-177.969,7.452,148.818
C08514=1147.651,210.936,-63.586,-177.971,7.450,148.819
C08515=1147.655,210.688,-63.562,-177.974,7.447,148.819
C08516=1147.659,210.439,-63.536,-177.977,7.444,148.819
C08517=1147.664,210.191,-63.511,-177.979,7.442,148.819
C08518=1147.669,209.920,-63.484,-177.982,7.439,148.819
C08519=1147.674,209.649,-63.458,-177.986,7.437,148.819
C08520=1147.679,209.379,-63.431,-177.988,7.434,148.820
C08521=1147.684,209.108,-63.404,-177.992,7.431,148.820
C08522=1147.688,208.859,-63.379,-177.994,7.428,148.820
C08523=1147.693,208.611,-63.355,-177.998,7.426,148.820
C08524=1147.698,208.362,-63.330,-178.000,7.424,148.820
C08525=1147.701,208.113,-63.305,-178.003,7.421,148.821
C08526=1147.706,207.865,-63.280,-178.005,7.419,148.821
C08527=1147.711,207.615,-63.255,-178.008,7.416,148.821
C08528=1147.715,207.367,-63.231,-178.011,7.414,148.821
C08529=1147.721,207.118,-63.206,-178.014,7.412,148.821
C08530=1147.724,206.869,-63.182,-178.016,7.409,148.822
C08531=1147.729,206.621,-63.157,-178.020,7.406,148.822
C08532=1147.734,206.372,-63.133,-178.022,7.404,148.822
C08533=1147.738,206.123,-63.108,-178.025,7.401,148.822
C08534=1147.742,205.875,-63.083,-178.028,7.398,148.822
C08535=1147.748,205.626,-63.059,-178.030,7.396,148.823
C08536=1147.751,205.377,-63.034,-178.033,7.394,148.823
C08537=1147.757,205.128,-63.010,-178.036,7.392,148.823
C08538=1147.761,204.880,-62.986,-178.039,7.389,148.823
C08539=1147.766,204.631,-62.961,-178.042,7.386,148.823
C08540=1147.770,204.382,-62.937,-178.044,7.385,148.824
C08541=1147.774,204.133,-62.912,-178.047,7.382,148.824
C08542=1147.779,203.885,-62.888,-178.050,7.379,148.824
C08543=1147.783,203.636,-62.863,-178.053,7.377,148.824
C08544=1147.788,203.387,-62.839,-178.055,7.374,148.824
C08545=1147.793,203.138,-62.815,-178.058,7.372,148.825
C08546=1147.797,202.889,-62.790,-178.061,7.369,148.825
C08547=1147.802,202.641,-62.765,-178.064,7.367,148.825
C08548=1147.806,202.392,-62.741,-178.066,7.365,148.825
C08549=1147.811,202.143,-62.717,-178.069,7.362,148.825
C08550=1147.815,201.894,-62.693,-178.072,7.360,148.826
C08551=1147.820,201.645,-62.669,-178.075,7.357,148.826
C08552=1147.825,201.397,-62.644,-178.078,7.355,148.826
C08553=1147.829,201.148,-62.620,-178.080,7.352,148.826
C08554=1147.833,200.899,-62.596,-178.083,7.350,148.827
C08555=1147.838,200.650,-62.572,-178.086,7.348,148.827
C08556=1147.843,200.401,-62.548,-178.089,7.345,148.827
C08557=1147.847,200.153,-62.524,-178.092,7.342,148.827
C08558=1147.852,199.904,-62.500,-178.094,7.341,148.828
C08559=1147.856,199.655,-62.475,-178.097,7.338,148.828
C08560=1147.861,199.406,-62.451,-178.100,7.336,148.828
C08561=1147.865,199.158,-62.427,-178.103,7.333,148.828
C08562=1147.870,198.909,-62.402,-178.105,7.331,148.829
C08563=1147.875,198.660,-62.378,-178.108,7.328,148.829
C08564=1147.879,198.411,-62.355,-178.111,7.325,148.829
C08565=1147.883,198.162,-62.331,-178.114,7.324,148.829
C08566=1147.888,197.914,-62.306,-178.117,7.321,148.829
C08567=1147.893,197.665,-62.283,-178.119,7.319,148.830
C08568=1147.897,197.416,-62.258,-178.122,7.316,148.830
C08569=1147.902,197.168,-62.234,-178.125,7.314,148.830
C08570=1147.907,196.919,-62.211,-178.128,7.311,148.830
C08571=1147.910,196.670,-62.187,-178.131,7.309,148.830
C08572=1147.916,196.420,-62.163,-178.133,7.307,148.831
C08573=1147.920,196.172,-62.139,-178.136,7.304,148.831
C08574=1147.925,195.923,-62.115,-178.138,7.302,148.831
C08575=1147.929,195.674,-62.091,-178.142,7.300,148.831
C08576=1147.934,195.426,-62.067,-178.144,7.298,148.832
C08577=1147.938,195.177,-62.044,-178.147,7.295,148.832
C08578=1147.944,194.928,-62.019,-178.150,7.293,148.832
C08579=1147.948,194.678,-61.995,-178.153,7.290,148.832
C08580=1147.952,194.430,-61.971,-178.155,7.289,148.833
C08581=1147.957,194.181,-61.948,-178.158,7.286,148.833
C08582=1147.961,193.933,-61.924,-178.162,7.283,148.833
C08583=1147.966,193.684,-61.900,-178.164,7.281,148.833
C08584=1147.970,193.435,-61.876,-178.167,7.278,148.834
C08585=1147.975,193.186,-61.853,-178.169,7.276,148.834
C08586=1147.980,192.937,-61.830,-178.172,7.274,148.834
C08587=1147.984,192.689,-61.806,-178.175,7.272,148.834
C08588=1147.989,192.440,-61.782,-178.178,7.269,148.835
C08589=1147.993,192.191,-61.758,-178.180,7.267,148.835
C08590=1147.998,191.942,-61.735,-178.183,7.264,148.835
C08591=1148.002,191.693,-61.711,-178.186,7.262,148.835
C08592=1148.007,191.445,-61.687,-178.189,7.260,148.835
C08593=1148.012,191.196,-61.664,-178.192,7.258,148.836
C08594=1148.016,190.947,-61.641,-178.194,7.255,148.836
C08595=1148.021,190.698,-61.617,-178.197,7.253,148.836
C08596=1148.025,190.449,-61.593,-178.200,7.251,148.836
C08597=1148.030,190.200,-61.570,-178.203,7.249,148.837
C08598=1148.035,189.951,-61.546,-178.205,7.246,148.837
C08599=1148.039,189.703,-61.522,-178.208,7.244,148.837
C08600=1148.044,189.454,-61.499,-178.211,7.241,148.837
C08601=1148.049,189.205,-61.476,-178.214,7.239,148.838
C08602=1148.053,188.956,-61.452,-178.217,7.237,148.838
C08603=1148.058,188.707,-61.428,-178.219,7.235,148.838
C08604=1148.062,188.458,-61.405,-178.222,7.232,148.839
C08605=1148.067,188.209,-61.382,-178.225,7.230,148.839
C08606=1148.072,187.960,-61.358,-178.228,7.228,148.839
C08607=1148.076,187.711,-61.335,-178.230,7.226,148.839
C08608=1148.081,187.462,-61.311,-178.233,7.223,148.839
C08609=1148.085,187.214,-61.288,-178.236,7.221,148.840
C08610=1148.089,186.965,-61.265,-178.239,7.218,148.840
C08611=1148.094,186.716,-61.241,-178.242,7.217,148.840
C08612=1148.099,186.467,-61.218,-178.244,7.214,148.840
C08613=1148.104,186.218,-61.195,-178.247,7.212,148.841
C08614=1148.108,185.969,-61.171,-178.250,7.209,148.841
C08615=1148.114,185.721,-61.148,-178.253,7.207,148.841
C08616=1148.118,185.472,-61.125,-178.256,7.205,148.842
C08617=1148.122,185.223,-61.102,-178.258,7.203,148.842
C08618=1148.127,184.974,-61.079,-178.261,7.200,148.842
C08619=1148.132,184.725,-61.055,-178.264,7.198,148.842
C08620=1148.136,184.476,-61.033,-178.266,7.196,148.843
C08621=1148.140,184.227,-61.009,-178.270,7.194,148.843
C08622=1148.145,183.958,-60.983,-178.273,7.191,148.843
C08623=1148.151,183.688,-60.958,-178.275,7.189,148.843
C08624=1148.155,183.419,-60.934,-178.278,7.187,148.844
C08625=1148.161,183.149,-60.909,-178.282,7.184,148.844
C08626=1148.165,182.900,-60.886,-178.284,7.182,148.844
C08627=1148.170,182.651,-60.862,-178.287,7.179,148.845
C08628=1148.174,182.402,-60.839,-178.290,7.178,148.845
C08629=1148.179,182.153,-60.816,-178.293,7.175,148.845
C08630=1148.184,181.905,-60.793,-178.295,7.173,148.845
C08631=1148.188,181.656,-60.770,-178.299,7.170,148.846
C08632=1148.193,181.406,-60.748,-178.301,7.168,148.846
C08633=1148.198,181.157,-60.724,-178.303,7.167,148.846
C08634=1148.202,180.909,-60.702,-178.307,7.164,148.847
C08635=1148.206,180.660,-60.678,-178.309,7.162,148.847
C08636=1148.212,180.411,-60.655,-178.312,7.159,148.847
C08637=1148.216,180.162,-60.633,-178.315,7.158,148.847
C08638=1148.221,179.913,-60.610,-178.318,7.155,148.848
C08639=1148.225,179.664,-60.586,-178.320,7.153,148.848
C08640=1148.229,179.415,-60.564,-178.324,7.150,148.848
C08641=1148.234,179.167,-60.541,-178.326,7.148,148.848
C08642=1148.239,178.917,-60.519,-178.329,7.147,148.849
C08643=1148.243,178.668,-60.495,-178.332,7.144,148.849
C08644=1148.248,178.419,-60.472,-178.334,7.142,148.849
C08645=1148.253,178.171,-60.450,-178.337,7.139,148.850
C08646=1148.258,177.922,-60.427,-178.340,7.138,148.850
C08647=1148.262,177.673,-60.404,-178.342,7.136,148.850
C08648=1148.267,177.423,-60.382,-178.346,7.133,148.850
C08649=1148.271,177.175,-60.359,-178.348,7.131,148.851
C08650=1148.276,176.926,-60.336,-178.351,7.128,148.851
C08651=1148.280,176.677,-60.314,-178.354,7.127,148.851
C08652=1148.286,176.429,-60.291,-178.357,7.125,148.852
C08653=1148.290,176.179,-60.269,-178.359,7.122,148.852
C08654=1148.294,175.930,-60.245,-178.362,7.120,148.852
C08655=1148.298,175.681,-60.223,-178.365,7.118,148.853
C08656=1148.304,175.433,-60.200,-178.368,7.116,148.853
C08657=1148.308,175.184,-60.178,-178.370,7.114,148.853
C08658=1148.313,174.934,-60.155,-178.374,7.111,148.853
C08659=1148.318,174.686,-60.132,-178.376,7.109,148.854
C08660=1148.323,174.436,-60.110,-178.379,7.107,148.854
C08661=1148.327,174.188,-60.087,-178.382,7.105,148.854
C08662=1148.332,173.939,-60.065,-178.384,7.103,148.855
C08663=1148.336,173.690,-60.042,-178.387,7.100,148.855
C08664=1148.340,173.441,-60.020,-178.390,7.099,148.855
C08665=1148.346,173.192,-59.997,-178.393,7.097,148.855
C08666=1148.350,172.943,-59.975,-178.395,7.094,148.856
C08667=1148.355,172.694,-59.952,-178.398,7.092,148.856
C08668=1148.360,172.445,-59.930,-178.401,7.090,148.856
C08669=1148.364,172.196,-59.908,-178.404,7.088,148.857
C08670=1148.368,171.947,-59.884,-178.406,7.086,148.857
C08671=1148.373,171.698,-59.863,-178.410,7.083,148.857
C08672=1148.377,171.450,-59.840,-178.412,7.082,148.858
C08673=1148.383,171.201,-59.818,-178.415,7.080,148.858
C08674=1148.387,170.951,-59.796,-178.418,7.077,148.858
C08675=1148.392,170.702,-59.772,-178.421,7.075,148.858
C08676=1148.397,170.454,-59.751,-178.423,7.074,148.859
C08677=1148.401,170.204,-59.729,-178.426,7.071,148.859
C08678=1148.406,169.956,-59.707,-178.429,7.069,148.859
C08679=1148.411,169.707,-59.684,-178.432,7.066,148.860
C08680=1148.415,169.458,-59.662,-178.435,7.065,148.860
C08681=1148.420,169.209,-59.640,-178.437,7.063,148.860
C08682=1148.424,168.960,-59.616,-178.440,7.060,148.861
C08683=1148.429,168.711,-59.595,-178.443,7.058,148.861
C08684=1148.434,168.462,-59.573,-178.446,7.057,148.861
C08685=1148.438,168.213,-59.551,-178.448,7.054,148.861
C08686=1148.443,167.963,-59.528,-178.451,7.052,148.862
C08687=1148.448,167.715,-59.506,-178.454,7.050,148.862
C08688=1148.452,167.466,-59.484,-178.457,7.048,148.862
C08689=1148.457,167.217,-59.462,-178.459,7.046,148.863
C08690=1148.462,166.968,-59.440,-178.462,7.044,148.863
C08691=1148.467,166.719,-59.418,-178.465,7.041,148.863
C08692=1148.471,166.470,-59.396,-178.468,7.040,148.864
C08693=1148.476,166.221,-59.374,-178.470,7.037,148.864
C08694=1148.480,165.972,-59.351,-178.474,7.035,148.864
C08695=1148.486,165.723,-59.329,-178.476,7.033,148.865
C08696=1148.490,165.474,-59.307,-178.479,7.031,148.865
C08697=1148.495,165.225,-59.285,-178.481,7.029,148.865
C08698=1148.499,164.976,-59.263,-178.484,7.027,148.865
C08699=1148.504,164.727,-59.242,-178.487,7.025,148.866
C08700=1148.508,164.478,-59.220,-178.490,7.023,148.866
C08701=1148.513,164.230,-59.198,-178.493,7.021,148.867
C08702=1148.517,163.980,-59.176,-178.495,7.019,148.867
C08703=1148.523,163.731,-59.154,-178.498,7.017,148.867
C08704=1148.527,163.482,-59.132,-178.501,7.014,148.867
C08705=1148.532,163.233,-59.110,-178.504,7.013,148.868
C08706=1148.536,162.984,-59.088,-178.507,7.011,148.868
C08707=1148.541,162.735,-59.066,-178.510,7.008,148.868
C08708=1148.546,162.487,-59.045,-178.512,7.006,148.869
C08709=1148.550,162.237,-59.022,-178.515,7.005,148.869
C08710=1148.555,161.989,-59.001,-178.518,7.003,148.869
C08711=1148.560,161.739,-58.979,-178.521,7.000,148.870
C08712=1148.565,161.490,-58.958,-178.523,6.998,148.870
C08713=1148.569,161.241,-58.936,-178.526,6.997,148.870
C08714=1148.574,160.992,-58.914,-178.529,6.994,148.871
C08715=1148.579,160.743,-58.892,-178.532,6.992,148.871
C08716=1148.583,160.494,-58.870,-178.535,6.991,148.871
C08717=1148.588,160.245,-58.849,-178.537,6.989,148.872
C08718=1148.593,159.996,-58.828,-178.540,6.986,148.872
C08719=1148.597,159.747,-58.806,-178.543,6.984,148.872
C08720=1148.602,159.498,-58.784,-178.546,6.983,148.873
C08721=1148.606,159.249,-58.762,-178.548,6.981,148.873
C08722=1148.611,159.000,-58.740,-178.552,6.978,148.873
C08723=1148.617,158.751,-58.719,-178.554,6.976,148.874
C08724=1148.621,158.502,-58.697,-178.556,6.974,148.874
C08725=1148.626,158.253,-58.676,-178.560,6.972,148.874
C08726=1148.630,157.984,-58.653,-178.562,6.970,148.875
C08727=1148.636,157.715,-58.629,-178.566,6.968,148.875
C08728=1148.640,157.446,-58.606,-178.568,6.966,148.875
C08729=1148.646,157.177,-58.583,-178.572,6.963,148.876
C08730=1148.651,156.928,-58.561,-178.574,6.962,148.876
C08731=1148.656,156.679,-58.540,-178.577,6.960,148.877
C08732=1148.660,156.430,-58.518,-178.579,6.958,148.877
C08733=1148.664,156.181,-58.497,-178.583,6.955,148.877
C08734=1148.669,155.932,-58.476,-178.585,6.954,148.878
C08735=1148.674,155.683,-58.454,-178.588,6.952,148.878
C08736=1148.679,155.434,-58.432,-178.591,6.950,148.878
C08737=1148.684,155.185,-58.411,-178.594,6.948,148.879
C08738=1148.689,154.936,-58.389,-178.597,6.946,148.879
C08739=1148.692,154.686,-58.369,-178.599,6.944,148.879
C08740=1148.697,154.438,-58.347,-178.602,6.942,148.880
C08741=1148.702,154.189,-58.326,-178.604,6.940,148.880
C08742=1148.707,153.940,-58.304,-178.608,6.938,148.880
C08743=1148.712,153.691,-58.282,-178.610,6.936,148.881
C08744=1148.716,153.442,-58.262,-178.613,6.934,148.881
C08745=1148.721,153.193,-58.240,-178.616,6.933,148.881
C08746=1148.726,152.944,-58.219,-178.619,6.930,148.882
C08747=1148.731,152.694,-58.198,-178.621,6.928,148.882
C08748=1148.736,152.445,-58.176,-178.624,6.926,148.882
C08749=1148.740,152.196,-58.156,-178.627,6.925,148.883
C08750=1148.745,151.947,-58.134,-178.629,6.923,148.883
C08751=1148.749,151.698,-58.113,-178.633,6.920,148.883
C08752=1148.754,151.449,-58.092,-178.635,6.919,148.884
C08753=1148.759,151.200,-58.071,-178.638,6.917,148.884
C08754=1148.764,150.951,-58.050,-178.641,6.915,148.885
C08755=1148.769,150.702,-58.028,-178.643,6.913,148.885
C08756=1148.773,150.453,-58.008,-178.646,6.911,148.885
C08757=1148.777,150.204,-57.986,-178.649,6.909,148.886
C08758=1148.783,149.954,-57.965,-178.652,6.907,148.886
C08759=1148.787,149.706,-57.944,-178.655,6.905,148.886
C08760=1148.792,149.457,-57.923,-178.657,6.904,148.887
C08761=1148.797,149.208,-57.902,-178.661,6.901,148.887
C08762=1148.802,148.959,-57.881,-178.663,6.899,148.887
C08763=1148.806,148.709,-57.859,-178.666,6.898,148.888
C08764=1148.811,148.460,-57.838,-178.669,6.896,148.888
C08765=1148.815,148.211,-57.818,-178.671,6.894,148.888
C08766=1148.821,147.962,-57.797,-178.674,6.891,148.889
C08767=1148.825,147.714,-57.776,-178.677,6.890,148.889
C08768=1148.830,147.464,-57.755,-178.680,6.888,148.889
C08769=1148.835,147.215,-57.734,-178.682,6.886,148.890
C08770=1148.839,146.965,-57.713,-178.685,6.885,148.890
C08771=1148.844,146.716,-57.692,-178.688,6.883,148.891
C08772=1148.848,146.468,-57.671,-178.691,6.880,148.891
C08773=1148.853,146.219,-57.650,-178.694,6.879,148.891
C08774=1148.858,145.970,-57.630,-178.696,6.877,148.892
C08775=1148.863,145.720,-57.609,-178.699,6.875,148.892
C08776=1148.867,145.471,-57.589,-178.702,6.873,148.893
C08777=1148.873,145.222,-57.568,-178.704,6.871,148.893
C08778=1148.877,144.973,-57.547,-178.707,6.869,148.893
C08779=1148.882,144.725,-57.526,-178.710,6.867,148.893
C08780=1148.886,144.476,-57.505,-178.713,6.865,148.894
C08781=1148.892,144.226,-57.484,-178.716,6.864,148.894
C08782=1148.895,143.977,-57.463,-178.718,6.862,148.895
C08783=1148.901,143.727,-57.442,-178.721,6.860,148.895
C08784=1148.905,143.478,-57.422,-178.724,6.859,148.895
C08785=1148.910,143.229,-57.401,-178.727,6.856,148.896
C08786=1148.915,142.980,-57.381,-178.730,6.854,148.896
C08787=1148.920,142.731,-57.360,-178.732,6.853,148.897
C08788=1148.924,142.482,-57.339,-178.735,6.851,148.897
C08789=1148.929,142.233,-57.318,-178.738,6.849,148.897
C08790=1148.934,141.984,-57.298,-178.741,6.847,148.898
C08791=1148.938,141.735,-57.278,-178.743,6.846,148.898
C08792=1148.943,141.486,-57.257,-178.747,6.843,148.898
C08793=1148.948,141.237,-57.236,-178.749,6.841,148.899
C08794=1148.953,140.987,-57.215,-178.752,6.840,148.899
C08795=1148.958,140.738,-57.195,-178.754,6.838,148.899
C08796=1148.962,140.490,-57.175,-178.757,6.836,148.900
C08797=1148.967,140.240,-57.154,-178.760,6.834,148.900
C08798=1148.972,139.991,-57.134,-178.762,6.833,148.901
C08799=1148.976,139.742,-57.114,-178.765,6.831,148.901
C08800=1148.981,139.492,-57.093,-178.768,6.828,148.901
C08801=1148.986,139.244,-57.072,-178.771,6.827,148.902
C08802=1148.990,138.995,-57.052,-178.774,6.825,148.902
C08803=1148.996,138.745,-57.031,-178.776,6.823,148.903
C08804=1149.000,138.496,-57.011,-178.779,6.821,148.903
C08805=1149.005,138.247,-56.991,-178.782,6.820,148.903
C08806=1149.010,137.998,-56.970,-178.785,6.818,148.904
C08807=1149.015,137.749,-56.950,-178.787,6.816,148.904
C08808=1149.019,137.500,-56.930,-178.790,6.815,148.904
C08809=1149.024,137.251,-56.909,-178.793,6.812,148.905
C08810=1149.029,137.002,-56.889,-178.796,6.810,148.905
C08811=1149.034,136.753,-56.869,-178.799,6.809,148.906
C08812=1149.038,136.504,-56.848,-178.801,6.807,148.906
C08813=1149.043,136.254,-56.829,-178.804,6.805,148.906
C08814=1149.048,136.005,-56.808,-178.807,6.804,148.907
C08815=1149.053,135.756,-56.787,-178.810,6.802,148.907
C08816=1149.057,135.507,-56.767,-178.812,6.800,148.908
C08817=1149.062,135.257,-56.747,-178.815,6.798,148.908
C08818=1149.067,135.009,-56.727,-178.818,6.797,148.908
C08819=1149.072,134.760,-56.706,-178.820,6.795,148.909
C08820=1149.077,134.510,-56.687,-178.823,6.793,148.909
C08821=1149.081,134.261,-56.666,-178.826,6.791,148.910
C08822=1149.086,134.012,-56.647,-178.829,6.789,148.910
C08823=1149.090,133.763,-56.626,-178.832,6.787,148.910
C08824=1149.095,133.514,-56.605,-178.835,6.786,148.911
C08825=1149.101,133.265,-56.586,-178.837,6.784,148.911
C08826=1149.105,133.016,-56.566,-178.840,6.782,148.912
C08827=1149.110,132.766,-56.546,-178.843,6.780,148.912
C08828=1149.114,132.517,-56.526,-178.845,6.779,148.912
C08829=1149.119,132.268,-56.506,-178.848,6.777,148.913
C08830=1149.124,131.999,-56.484,-178.851,6.775,148.913
C08831=1149.129,131.731,-56.462,-178.855,6.773,148.914
C08832=1149.135,131.462,-56.441,-178.857,6.771,148.914
C08833=1149.140,131.194,-56.419,-178.860,6.770,148.914
C08834=1149.145,130.945,-56.400,-178.863,6.768,148.915
C08835=1149.149,130.696,-56.379,-178.866,6.766,148.915
C08836=1149.154,130.446,-56.360,-178.868,6.765,148.916
C08837=1149.159,130.197,-56.339,-178.871,6.763,148.916
C08838=1149.163,129.948,-56.320,-178.874,6.760,148.916
C08839=1149.169,129.699,-56.300,-178.877,6.759,148.917
C08840=1149.174,129.450,-56.279,-178.880,6.757,148.917
C08841=1149.179,129.200,-56.260,-178.882,6.755,148.918
C08842=1149.183,128.951,-56.239,-178.885,6.754,148.918
C08843=1149.188,128.702,-56.220,-178.888,6.752,148.918
C08844=1149.193,128.453,-56.200,-178.891,6.750,148.919
C08845=1149.198,128.204,-56.180,-178.893,6.748,148.919
C08846=1149.202,127.954,-56.160,-178.896,6.747,148.920
C08847=1149.208,127.705,-56.141,-178.899,6.745,148.920
C08848=1149.212,127.456,-56.121,-178.901,6.743,148.920
C08849=1149.217,127.207,-56.101,-178.905,6.742,148.921
C08850=1149.221,126.958,-56.082,-178.907,6.740,148.921
C08851=1149.226,126.709,-56.062,-178.910,6.739,148.922
C08852=1149.231,126.460,-56.042,-178.913,6.737,148.922
C08853=1149.235,126.210,-56.023,-178.916,6.735,148.923
C08854=1149.241,125.961,-56.003,-178.918,6.733,148.923
C08855=1149.245,125.712,-55.983,-178.921,6.732,148.923
C08856=1149.250,125.463,-55.963,-178.924,6.730,148.924
C08857=1149.255,125.214,-55.944,-178.926,6.728,148.924
C08858=1149.260,124.964,-55.924,-178.929,6.727,148.925
C08859=1149.264,124.715,-55.904,-178.932,6.725,148.925
C08860=1149.270,124.466,-55.885,-178.935,6.723,148.925
C08861=1149.274,124.217,-55.866,-178.937,6.722,148.926
C08862=1149.279,123.968,-55.846,-178.940,6.720,148.926
C08863=1149.284,123.719,-55.827,-178.943,6.718,148.927
C08864=1149.289,123.469,-55.807,-178.945,6.716,148.927
C08865=1149.293,123.220,-55.787,-178.949,6.715,148.928
C08866=1149.298,122.971,-55.767,-178.951,6.713,148.928
C08867=1149.303,122.722,-55.748,-178.954,6.712,148.928
C08868=1149.307,122.473,-55.729,-178.957,6.710,148.929
C08869=1149.312,122.224,-55.709,-178.960,6.708,148.929
C08870=1149.317,121.974,-55.690,-178.962,6.707,148.930
C08871=1149.322,121.725,-55.670,-178.965,6.705,148.930
C08872=1149.327,121.476,-55.651,-178.968,6.703,148.930
C08873=1149.331,121.226,-55.632,-178.970,6.701,148.931
C08874=1149.337,120.978,-55.612,-178.973,6.700,148.931
C08875=1149.341,120.728,-55.593,-178.976,6.698,148.932
C08876=1149.346,120.478,-55.573,-178.979,6.696,148.932
C08877=1149.351,120.230,-55.554,-178.982,6.695,148.933
C08878=1149.356,119.980,-55.535,-178.984,6.693,148.933
C08879=1149.361,119.731,-55.515,-178.987,6.692,148.933
C08880=1149.366,119.482,-55.496,-178.990,6.690,148.934
C08881=1149.370,119.233,-55.477,-178.993,6.688,148.934
C08882=1149.375,118.984,-55.457,-178.995,6.687,148.935
C08883=1149.380,118.734,-55.438,-178.998,6.685,148.935
C08884=1149.384,118.486,-55.419,-179.001,6.683,148.935
C08885=1149.389,118.236,-55.399,-179.003,6.682,148.936
C08886=1149.394,117.987,-55.380,-179.006,6.681,148.936
C08887=1149.399,117.738,-55.361,-179.009,6.679,148.937
C08888=1149.404,117.489,-55.342,-179.012,6.677,148.937
C08889=1149.408,117.240,-55.322,-179.014,6.676,148.938
C08890=1149.414,116.990,-55.304,-179.017,6.674,148.938
C08891=1149.418,116.741,-55.285,-179.020,6.672,148.939
C08892=1149.423,116.492,-55.265,-179.022,6.671,148.939
C08893=1149.428,116.242,-55.246,-179.025,6.669,148.939
C08894=1149.433,115.994,-55.227,-179.028,6.667,148.940
C08895=1149.438,115.744,-55.207,-179.031,6.666,148.940
C08896=1149.442,115.495,-55.189,-179.034,6.664,148.941
C08897=1149.447,115.245,-55.170,-179.037,6.663,148.941
C08898=1149.453,114.997,-55.150,-179.039,6.661,148.942
C08899=1149.457,114.747,-55.131,-179.042,6.659,148.942
C08900=1149.462,114.498,-55.113,-179.045,6.657,148.942
C08901=1149.466,114.249,-55.094,-179.047,6.656,148.943
C08902=1149.472,114.000,-55.074,-179.050,6.655,148.943
C08903=1149.476,113.750,-55.055,-179.053,6.654,148.944
C08904=1149.481,113.501,-55.037,-179.056,6.652,148.944
C08905=1149.486,113.251,-55.017,-179.058,6.650,148.945
C08906=1149.491,113.003,-54.998,-179.061,6.648,148.945
C08907=1149.496,112.753,-54.979,-179.064,6.647,148.945
C08908=1149.500,112.504,-54.961,-179.066,6.645,148.946
C08909=1149.506,112.255,-54.941,-179.069,6.643,148.946
C08910=1149.510,112.005,-54.923,-179.072,6.642,148.947
C08911=1149.515,111.757,-54.904,-179.075,6.640,148.947
C08912=1149.519,111.507,-54.885,-179.078,6.639,148.948
C08913=1149.525,111.258,-54.866,-179.080,6.638,148.948
C08914=1149.529,111.009,-54.847,-179.083,6.636,148.949
C08915=1149.535,110.759,-54.828,-179.085,6.634,148.949
C08916=1149.539,110.510,-54.810,-179.088,6.633,148.949
C08917=1149.544,110.260,-54.791,-179.091,6.631,148.950
C08918=1149.549,110.012,-54.772,-179.094,6.630,148.950
C08919=1149.554,109.763,-54.753,-179.097,6.628,148.951
C08920=1149.558,109.513,-54.735,-179.100,6.626,148.951
C08921=1149.563,109.264,-54.716,-179.102,6.625,148.952
C08922=1149.568,109.014,-54.697,-179.105,6.623,148.952
C08923=1149.573,108.766,-54.678,-179.107,6.622,148.952
C08924=1149.578,108.516,-54.660,-179.110,6.621,148.953
C08925=1149.582,108.267,-54.641,-179.113,6.619,148.954
C08926=1149.588,108.017,-54.622,-179.116,6.617,148.954
C08927=1149.593,107.769,-54.603,-179.118,6.616,148.954
C08928=1149.597,107.519,-54.585,-179.121,6.614,148.955
C08929=1149.603,107.270,-54.566,-179.124,6.612,148.955
C08930=1149.607,107.021,-54.548,-179.127,6.611,148.956
C08931=1149.611,106.771,-54.529,-179.129,6.610,148.956
C08932=1149.617,106.522,-54.510,-179.132,6.608,148.957
C08933=1149.622,106.273,-54.492,-179.135,6.607,148.957
C08934=1149.627,106.004,-54.472,-179.137,6.605,148.957
C08935=1149.632,105.736,-54.452,-179.141,6.604,148.958
C08936=1149.638,105.468,-54.432,-179.143,6.602,148.958
C08937=1149.643,105.199,-54.412,-179.147,6.601,148.959
C08938=1149.647,104.950,-54.393,-179.149,6.599,148.960
C08939=1149.652,104.701,-54.374,-179.152,6.597,148.960
C08940=1149.657,104.451,-54.357,-179.155,6.595,148.960
C08941=1149.662,104.202,-54.339,-179.158,6.594,148.961
C08942=1149.666,103.953,-54.319,-179.160,6.592,148.961
C08943=1149.672,103.703,-54.301,-179.163,6.591,148.962
C08944=1149.677,103.454,-54.283,-179.166,6.590,148.962
C08945=1149.681,103.205,-54.264,-179.168,6.588,148.963
C08946=1149.686,102.956,-54.246,-179.171,6.587,148.963
C08947=1149.691,102.706,-54.227,-179.174,6.585,148.963
C08948=1149.696,102.457,-54.209,-179.177,6.584,148.964
C08949=1149.700,102.208,-54.190,-179.180,6.582,148.964
C08950=1149.705,101.959,-54.172,-179.182,6.581,148.965
C08951=1149.711,101.709,-54.154,-179.185,6.579,148.965
C08952=1149.716,101.460,-54.136,-179.187,6.578,148.966
C08953=1149.721,101.211,-54.118,-179.191,6.576,148.966
C08954=1149.725,100.962,-54.099,-179.193,6.575,148.967
C08955=1149.729,100.713,-54.081,-179.196,6.573,148.967
C08956=1149.735,100.463,-54.062,-179.198,6.572,148.968
C08957=1149.740,100.214,-54.044,-179.201,6.570,148.968
C08958=1149.745,99.965,-54.026,-179.204,6.569,148.969
C08959=1149.749,99.715,-54.008,-179.207,6.567,148.969
C08960=1149.754,99.466,-53.990,-179.210,6.566,148.970
C08961=1149.759,99.216,-53.972,-179.212,6.564,148.970
C08962=1149.764,98.967,-53.954,-179.214,6.563,148.970
C08963=1149.769,98.719,-53.935,-179.218,6.562,148.971
C08964=1149.774,98.469,-53.916,-179.220,6.560,148.971
C08965=1149.779,98.219,-53.898,-179.223,6.558,148.972
C08966=1149.783,97.970,-53.880,-179.226,6.557,148.972
C08967=1149.788,97.721,-53.862,-179.228,6.556,148.973
C08968=1149.793,97.472,-53.844,-179.231,6.554,148.973
C08969=1149.798,97.223,-53.826,-179.234,6.553,148.974
C08970=1149.803,96.973,-53.808,-179.237,6.551,148.974
C08971=1149.807,96.724,-53.790,-179.239,6.549,148.975
C08972=1149.812,96.474,-53.772,-179.242,6.549,148.975
C08973=1149.817,96.225,-53.754,-179.245,6.547,148.976
C08974=1149.822,95.976,-53.736,-179.247,6.546,148.976
C08975=1149.827,95.727,-53.718,-179.250,6.544,148.976
C08976=1149.832,95.478,-53.700,-179.253,6.543,148.977
C08977=1149.837,95.228,-53.683,-179.255,6.542,148.977
C08978=1149.842,94.978,-53.665,-179.258,6.540,148.978
C08979=1149.846,94.729,-53.647,-179.261,6.538,148.978
C08980=1149.851,94.480,-53.629,-179.264,6.537,148.979
C08981=1149.856,94.231,-53.611,-179.266,6.536,148.979
C08982=1149.861,93.981,-53.593,-179.269,6.534,148.980
C08983=1149.866,93.732,-53.575,-179.272,6.533,148.980
C08984=1149.871,93.483,-53.557,-179.275,6.531,148.981
C08985=1149.876,93.234,-53.539,-179.278,6.530,148.981
C08986=1149.881,92.984,-53.521,-179.280,6.529,148.982
C08987=1149.886,92.735,-53.503,-179.283,6.527,148.982
C08988=1149.891,92.486,-53.485,-179.285,6.525,148.983
C08989=1149.896,92.237,-53.467,-179.289,6.524,148.983
C08990=1149.901,91.987,-53.449,-179.291,6.523,148.984
C08991=1149.906,91.738,-53.432,-179.293,6.522,148.984
C08992=1149.910,91.488,-53.414,-179.296,6.520,148.984
C08993=1149.915,91.238,-53.396,-179.299,6.519,148.985
C08994=1149.920,90.989,-53.378,-179.302,6.518,148.986
C08995=1149.925,90.739,-53.361,-179.304,6.516,148.986
C08996=1149.930,90.491,-53.343,-179.307,6.514,148.986
C08997=1149.934,90.241,-53.325,-179.310,6.513,148.987
C08998=1149.939,89.992,-53.307,-179.312,6.512,148.987
C08999=1149.945,89.742,-53.290,-179.315,6.510,148.988
C09000=1149.949,89.493,-53.272,-179.318,6.509,148.988
C09001=1149.954,89.244,-53.254,-179.321,6.507,148.989
C09002=1149.960,88.994,-53.237,-179.323,6.507,148.989
C09003=1149.964,88.745,-53.219,-179.326,6.505,148.990
C09004=1149.969,88.496,-53.201,-179.329,6.503,148.990
C09005=1149.974,88.247,-53.184,-179.332,6.502,148.991
C09006=1149.979,87.997,-53.166,-179.334,6.501,148.991
C09007=1149.984,87.748,-53.149,-179.337,6.499,148.992
C09008=1149.989,87.498,-53.131,-179.339,6.498,148.992
C09009=1149.993,87.250,-53.114,-179.342,6.497,148.993
C09010=1149.999,87.000,-53.097,-179.345,6.496,148.993
C09011=1150.004,86.751,-53.079,-179.348,6.494,148.994
C09012=1150.009,86.501,-53.061,-179.351,6.493,148.994
C09013=1150.013,86.253,-53.044,-179.353,6.492,148.995
C09014=1150.018,86.003,-53.026,-179.356,6.490,148.995
C09015=1150.023,85.754,-53.009,-179.358,6.488,148.996
C09016=1150.028,85.504,-52.991,-179.361,6.488,148.996
C09017=1150.033,85.255,-52.974,-179.364,6.486,148.997
C09018=1150.038,85.006,-52.956,-179.366,6.484,148.997
C09019=1150.043,84.756,-52.939,-179.369,6.483,148.997
C09020=1150.048,84.507,-52.921,-179.372,6.482,148.998
C09021=1150.052,84.257,-52.904,-179.375,6.481,148.999
C09022=1150.058,84.008,-52.887,-179.377,6.479,148.999
C09023=1150.063,83.759,-52.869,-179.380,6.478,149.000
C09024=1150.068,83.510,-52.853,-179.383,6.477,149.000
C09025=1150.072,83.260,-52.835,-179.385,6.475,149.000
C09026=1150.078,83.011,-52.817,-179.388,6.473,149.001
C09027=1150.082,82.762,-52.800,-179.391,6.473,149.002
C09028=1150.087,82.512,-52.783,-179.394,6.471,149.002
C09029=1150.092,82.262,-52.766,-179.396,6.470,149.002
C09030=1150.096,82.013,-52.748,-179.399,6.469,149.003
C09031=1150.102,81.763,-52.731,-179.402,6.467,149.003
C09032=1150.107,81.515,-52.713,-179.404,6.466,149.004
C09033=1150.112,81.266,-52.697,-179.407,6.465,149.005
C09034=1150.117,81.016,-52.679,-179.410,6.464,149.005
C09035=1150.121,80.767,-52.662,-179.412,6.462,149.005
C09036=1150.126,80.517,-52.645,-179.415,6.461,149.006
C09037=1150.131,80.267,-52.627,-179.418,6.460,149.006
C09038=1150.137,79.999,-52.610,-179.421,6.458,149.007
C09039=1150.142,79.731,-52.590,-179.424,6.457,149.008
C09040=1150.148,79.463,-52.572,-179.427,6.455,149.008
C09041=1150.152,79.194,-52.554,-179.430,6.454,149.009
C09042=1150.158,78.945,-52.537,-179.432,6.453,149.009
C09043=1150.162,78.695,-52.520,-179.435,6.451,149.009
C09044=1150.168,78.447,-52.502,-179.438,6.450,149.010
C09045=1150.172,78.197,-52.486,-179.440,6.449,149.011
C09046=1150.177,77.947,-52.468,-179.443,6.447,149.011
C09047=1150.182,77.698,-52.452,-179.445,6.446,149.011
C09048=1150.187,77.448,-52.434,-179.448,6.445,149.012
C09049=1150.192,77.200,-52.417,-179.451,6.443,149.012
C09050=1150.197,76.950,-52.400,-179.454,6.442,149.013
C09051=1150.202,76.701,-52.384,-179.456,6.441,149.014
C09052=1150.207,76.451,-52.366,-179.459,6.440,149.014
C09053=1150.212,76.202,-52.350,-179.461,6.439,149.014
C09054=1150.217,75.952,-52.333,-179.464,6.437,149.015
C09055=1150.222,75.703,-52.316,-179.467,6.436,149.016
C09056=1150.226,75.454,-52.298,-179.469,6.435,149.016
C09057=1150.231,75.205,-52.282,-179.472,6.434,149.017
C09058=1150.237,74.955,-52.264,-179.475,6.432,149.017
C09059=1150.241,74.706,-52.248,-179.477,6.431,149.017
C09060=1150.246,74.456,-52.231,-179.481,6.430,149.018
C09061=1150.251,74.207,-52.214,-179.483,6.428,149.019
C09062=1150.256,73.958,-52.198,-179.485,6.427,149.019
C09063=1150.261,73.708,-52.180,-179.489,6.426,149.020
C09064=1150.266,73.458,-52.164,-179.491,6.425,149.020
C09065=1150.271,73.209,-52.147,-179.494,6.423,149.020
C09066=1150.276,72.960,-52.130,-179.496,6.422,149.021
C09067=1150.280,72.710,-52.113,-179.499,6.421,149.022
C09068=1150.286,72.461,-52.096,-179.502,6.420,149.022
C09069=1150.291,72.212,-52.080,-179.504,6.418,149.022
C09070=1150.296,71.962,-52.063,-179.507,6.417,149.023
C09071=1150.301,71.713,-52.046,-179.510,6.416,149.024
C09072=1150.306,71.464,-52.030,-179.512,6.415,149.024
C09073=1150.311,71.214,-52.012,-179.515,6.414,149.025
C09074=1150.316,70.965,-51.996,-179.518,6.412,149.025
C09075=1150.320,70.715,-51.979,-179.520,6.411,149.025
C09076=1150.326,70.466,-51.962,-179.523,6.410,149.026
C09077=1150.331,70.217,-51.946,-179.525,6.409,149.027
C09078=1150.335,69.967,-51.929,-179.528,6.407,149.027
C09079=1150.340,69.717,-51.913,-179.531,6.406,149.028
C09080=1150.346,69.468,-51.896,-179.534,6.405,149.028
C09081=1150.350,69.219,-51.880,-179.537,6.404,149.029
C09082=1150.355,68.970,-51.863,-179.539,6.403,149.029
C09083=1150.360,68.720,-51.846,-179.542,6.401,149.030
C09084=1150.365,68.471,-51.829,-179.545,6.400,149.030
C09085=1150.370,68.222,-51.813,-179.547,6.399,149.031
C09086=1150.375,67.972,-51.797,-179.550,6.397,149.031
C09087=1150.380,67.722,-51.780,-179.552,6.397,149.032
C09088=1150.385,67.473,-51.764,-179.555,6.395,149.032
C09089=1150.390,67.224,-51.747,-179.558,6.394,149.033
C09090=1150.395,66.975,-51.731,-179.561,6.393,149.033
C09091=1150.400,66.725,-51.714,-179.563,6.391,149.034
C09092=1150.405,66.475,-51.697,-179.565,6.391,149.034
C09093=1150.410,66.226,-51.681,-179.569,6.389,149.035
C09094=1150.414,65.977,-51.664,-179.571,6.388,149.035
C09095=1150.420,65.727,-51.649,-179.574,6.387,149.036
C09096=1150.424,65.478,-51.632,-179.577,6.386,149.036
C09097=1150.430,65.229,-51.615,-179.579,6.385,149.037
C09098=1150.435,64.979,-51.599,-179.582,6.383,149.037
C09099=1150.439,64.729,-51.583,-179.584,6.382,149.038
C09100=1150.444,64.480,-51.566,-179.587,6.381,149.038
C09101=1150.449,64.230,-51.550,-179.590,6.380,149.039
C09102=1150.454,63.982,-51.534,-179.592,6.379,149.039
C09103=1150.459,63.732,-51.517,-179.595,6.377,149.040
C09104=1150.465,63.482,-51.501,-179.598,6.377,149.041
C09105=1150.469,63.233,-51.485,-179.601,6.375,149.041
C09106=1150.474,62.984,-51.468,-179.603,6.374,149.041
C09107=1150.479,62.734,-51.452,-179.606,6.373,149.042
C09108=1150.484,62.485,-51.436,-179.608,6.372,149.043
C09109=1150.489,62.235,-51.420,-179.611,6.370,149.043
C09110=1150.494,61.986,-51.404,-179.613,6.370,149.044
C09111=1150.499,61.737,-51.387,-179.616,6.368,149.044
C09112=1150.504,61.487,-51.371,-179.619,6.367,149.045
C09113=1150.509,61.238,-51.354,-179.622,6.366,149.045
C09114=1150.515,60.988,-51.339,-179.624,6.364,149.046
C09115=1150.519,60.739,-51.322,-179.627,6.364,149.046
C09116=1150.524,60.489,-51.306,-179.630,6.362,149.047
C09117=1150.529,60.240,-51.290,-179.632,6.361,149.047
C09118=1150.534,59.990,-51.274,-179.635,6.360,149.048
C09119=1150.539,59.741,-51.257,-179.637,6.359,149.048
C09120=1150.544,59.492,-51.242,-179.640,6.357,149.049
C09121=1150.549,59.243,-51.226,-179.643,6.357,149.049
C09122=1150.554,58.993,-51.210,-179.645,6.355,149.050
C09123=1150.559,58.744,-51.193,-179.648,6.355,149.050
C09124=1150.564,58.494,-51.177,-179.651,6.353,149.051
C09125=1150.569,58.244,-51.162,-179.653,6.352,149.051
C09126=1150.574,57.995,-51.145,-179.656,6.351,149.052
C09127=1150.579,57.745,-51.129,-179.659,6.349,149.052
C09128=1150.584,57.496,-51.113,-179.662,6.349,149.053
C09129=1150.589,57.247,-51.097,-179.664,6.347,149.054
C09130=1150.594,56.997,-51.082,-179.666,6.346,149.054
C09131=1150.599,56.748,-51.065,-179.670,6.345,149.055
C09132=1150.604,56.498,-51.049,-179.672,6.344,149.055
C09133=1150.608,56.249,-51.033,-179.675,6.343,149.056
C09134=1150.613,56.000,-51.018,-179.677,6.342,149.056
C09135=1150.619,55.750,-51.002,-179.680,6.340,149.057
C09136=1150.623,55.501,-50.985,-179.683,6.340,149.057
C09137=1150.629,55.251,-50.970,-179.685,6.338,149.058
C09138=1150.634,55.002,-50.954,-179.688,6.337,149.058
C09139=1150.638,54.753,-50.938,-179.691,6.336,149.059
C09140=1150.644,54.503,-50.922,-179.693,6.335,149.059
C09141=1150.649,54.253,-50.906,-179.696,6.334,149.060
C09142=1150.654,53.985,-50.889,-179.698,6.333,149.060
C09143=1150.660,53.716,-50.872,-179.702,6.332,149.061
C09144=1150.665,53.448,-50.855,-179.704,6.330,149.061
C09145=1150.670,53.179,-50.839,-179.707,6.330,149.062
C09146=1150.675,52.929,-50.823,-179.710,6.328,149.063
C09147=1150.680,52.680,-50.807,-179.712,6.328,149.063
C09148=1150.685,52.431,-50.791,-179.715,6.326,149.064
C09149=1150.690,52.181,-50.775,-179.717,6.325,149.064
C09150=1150.696,51.932,-50.759,-179.720,6.324,149.065
C09151=1150.700,51.683,-50.744,-179.723,6.323,149.065
